RoboDK station: main2.rdk

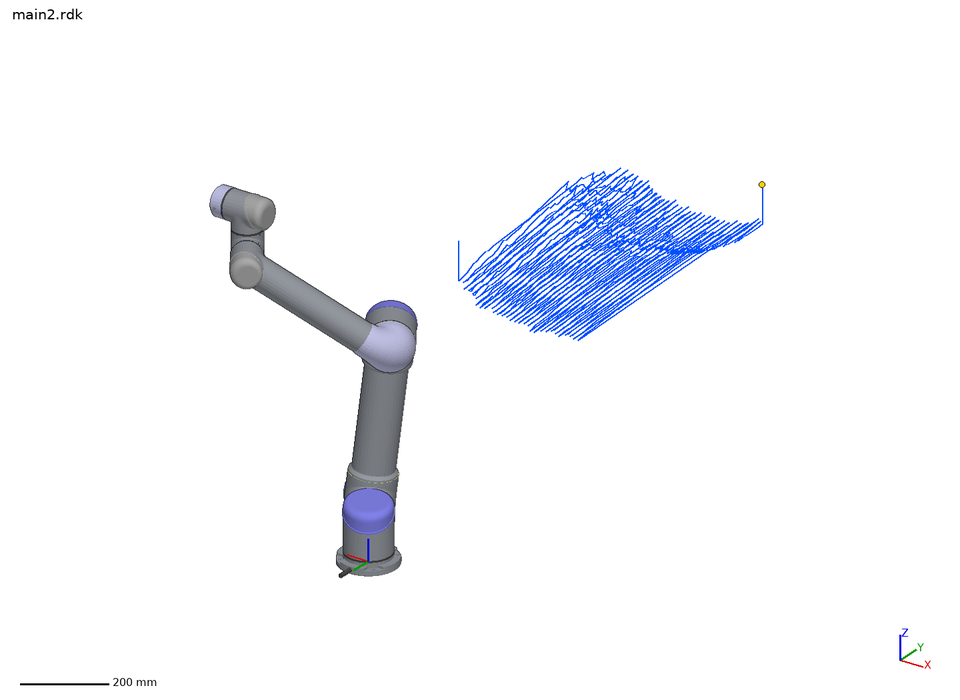
[picture v0: the station drawn from its stored meshes, robots at their saved joint values, targets as dots, program paths as lines]
Station main. Poses are relative to the parent item; angles as X-Y-Z fixed-axis rotations.
  - frame UR5 Base at (0, 0, 0) mm, rotated rx 0 ry 0 rz 180 deg
    - robot UR5: 6 axes, payload 5 kg, reach 850 mm, repeatability 0.1 mm, weight 18.4 kg
        modified DH rows (alpha deg, a mm, theta deg, d mm): 0, 0, 0, 89.2; 90, 0, 180, 0; 0, 425, 0, 0; 0, 392.43, 0, 109; -90, 0, 0, 93.65; 90, 0, 180, 82
        joint limits [-360, -360, -360, -360, -360, -360] to [360, 360, 360, 360, 360, 360]; home [0, -90, -90, 0, 90, 0]; saved at [33.979, -83.621, -61.636, -34.743, 56.021, -90]
  - frame Object at (-1200, -500, 400) mm, rotated rx -90 ry 0 rz -90 deg
    - object Curve at (0, 0, 0) mm
  - machining project AutoCurveFollow settings: rotZ(0) | rotX(0)*rotY(0) | rotz(0) | onStart | onPathStart | onApproach | onPoint | onRetract | onFinish | Extruder(%1) | default | default | OutOnMov(%1) | OutOffMov(%1) | onPathFinish | M_RunCode(%1)
  - program AutoCurveFollow (1423 instructions, listed below)
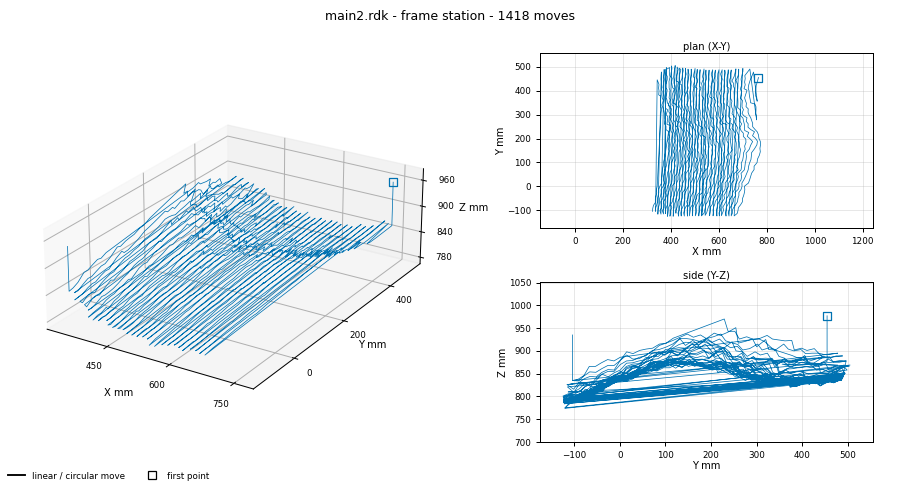
[picture p0: tool path of main2.rdk in frame station, 1418 of 1418 moves have a stored position in this frame; points joined in program order, loops and branches not executed]

--- program AutoCurveFollow (robot UR5) ---
  Set Ref.: UR5 Base
  Set Tool at (0, 0, 0) mm
  Set speed (1000.0 mm/s)
  MoveJ 1 to (-764.48, -454.56, 977) mm, rotated rx 180 ry 0 rz -90 deg; joints [-40.611, -86.577, -54.328, -39.095, 130.611, -90]
  MoveL 2 to (-764.48, -454.56, 977) mm, rotated rx 180 ry 0 rz -90 deg; joints [-40.611, -86.577, -54.328, -39.095, 130.611, -90]
  MoveL 3 to (-764.48, -454.56, 877) mm, rotated rx 180 ry 0 rz -90 deg; joints [-29.923, -94.985, -45.76, -39.255, 119.923, -90]
  MoveL 4 to (-764.48, -454.56, 877) mm, rotated rx 180 ry 0 rz -90 deg; joints [-29.923, -94.985, -45.76, -39.255, 119.923, -90]
  Set speed (50.0 mm/s)
  MoveL 5 to (-760.12, -438.29, 872) mm, rotated rx 180 ry 0 rz -90 deg; joints [-28.873, -93.22, -50.699, -36.081, 118.873, -90]
  MoveL 6 to (-754.89, -421.7, 866) mm, rotated rx 180 ry 0 rz -90 deg; joints [-27.622, -91.69, -55.258, -33.052, 117.622, -90]
  MoveL 7 to (-754.02, -407.65, 865) mm, rotated rx 180 ry 0 rz -90 deg; joints [-27.415, -90.512, -58.88, -30.609, 117.415, -90]
  MoveL 8 to (-752.27, -393.17, 863) mm, rotated rx 180 ry 0 rz -90 deg; joints [-27.002, -89.439, -62.378, -28.183, 117.002, -90]
  MoveL 9 to (-752.27, -379.64, 863) mm, rotated rx 180 ry 0 rz -90 deg; joints [-27.002, -88.514, -65.502, -25.984, 117.002, -90]
  MoveL 10 to (-756.63, -368.22, 868) mm, rotated rx 180 ry 0 rz -90 deg; joints [-28.038, -87.745, -68.081, -24.174, 118.038, -90]
  MoveL 11 to (-759.25, -355.84, 871) mm, rotated rx 180 ry 0 rz -90 deg; joints [-28.664, -87.014, -70.74, -22.246, 118.664, -90]
  MoveL 12 to (-743.88, -477.67, 869) mm, rotated rx 180 ry 0 rz -90 deg; joints [-26.18, -96.591, -39.404, -44.005, 116.18, -90]
  MoveL 13 to (-729.32, -441.6, 852) mm, rotated rx 180 ry 0 rz -90 deg; joints [-22.685, -92.557, -50.807, -36.636, 112.685, -90]
  MoveL 14 to (-724.19, -425.22, 846) mm, rotated rx 180 ry 0 rz -90 deg; joints [-21.483, -91.151, -55.197, -33.652, 111.483, -90]
  MoveL 15 to (-721.62, -410.5, 843) mm, rotated rx 180 ry 0 rz -90 deg; joints [-20.889, -89.985, -58.924, -31.091, 110.889, -90]
  MoveL 16 to (-725.04, -399.16, 847) mm, rotated rx 180 ry 0 rz -90 deg; joints [-21.682, -88.972, -61.84, -29.189, 111.682, -90]
  MoveL 17 to (-725.9, -386.34, 848) mm, rotated rx 180 ry 0 rz -90 deg; joints [-21.882, -88.028, -64.877, -27.095, 111.882, -90]
  MoveL 18 to (-727.61, -373.92, 850) mm, rotated rx 180 ry 0 rz -90 deg; joints [-22.282, -87.165, -67.716, -25.119, 112.282, -90]
  MoveL 19 to (-730.18, -361.86, 853) mm, rotated rx 180 ry 0 rz -90 deg; joints [-22.887, -86.368, -70.389, -23.243, 112.887, -90]
  MoveL 20 to (-731.89, -349.3, 855) mm, rotated rx 180 ry 0 rz -90 deg; joints [-23.292, -85.64, -73.039, -21.321, 113.292, -90]
  MoveL 21 to (-749.87, -344.14, 876) mm, rotated rx 180 ry 0 rz -90 deg; joints [-27.655, -84.997, -74.428, -20.575, 117.655, -90]
  MoveL 22 to (-754.15, -332.29, 881) mm, rotated rx 180 ry 0 rz -90 deg; joints [-28.72, -84.394, -76.805, -18.802, 118.72, -90]
  MoveL 23 to (-754.15, -318.48, 881) mm, rotated rx 180 ry 0 rz -90 deg; joints [-28.72, -83.813, -79.436, -16.751, 118.72, -90]
  MoveL 24 to (-753.29, -304.32, 880) mm, rotated rx 180 ry 0 rz -90 deg; joints [-28.506, -83.297, -82.034, -14.669, 118.506, -90]
  MoveL 25 to (-755.86, -291.51, 883) mm, rotated rx 180 ry 0 rz -90 deg; joints [-29.148, -82.862, -84.336, -12.802, 119.148, -90]
  MoveL 26 to (-756.72, -277.98, 884) mm, rotated rx 180 ry 0 rz -90 deg; joints [-29.363, -82.481, -86.682, -10.837, 119.363, -90]
  MoveL 27 to (-728.57, -490.16, 867) mm, rotated rx 180 ry 0 rz -90 deg; joints [-23.594, -97.07, -36.241, -46.688, 113.594, -90]
  MoveL 28 to (-707.56, -462.82, 842) mm, rotated rx 180 ry 0 rz -90 deg; joints [-18.545, -94.089, -45.181, -40.73, 108.545, -90]
  MoveL 29 to (-709.24, -450.69, 844) mm, rotated rx 180 ry 0 rz -90 deg; joints [-18.936, -92.582, -49.108, -38.31, 108.936, -90]
  MoveL 30 to (-706.72, -435.9, 841) mm, rotated rx 180 ry 0 rz -90 deg; joints [-18.351, -91.172, -53.282, -35.546, 108.351, -90]
  MoveL 31 to (-709.24, -424.22, 844) mm, rotated rx 180 ry 0 rz -90 deg; joints [-18.936, -89.957, -56.582, -33.46, 108.936, -90]
  MoveL 32 to (-704.2, -408.06, 838) mm, rotated rx 180 ry 0 rz -90 deg; joints [-17.77, -88.854, -60.455, -30.691, 107.77, -90]
  MoveL 33 to (-716.8, -401.99, 853) mm, rotated rx 180 ry 0 rz -90 deg; joints [-20.724, -87.803, -62.493, -29.704, 110.724, -90]
  MoveL 34 to (-711.76, -385.88, 847) mm, rotated rx 180 ry 0 rz -90 deg; joints [-19.527, -86.87, -66.047, -27.083, 109.527, -90]
  MoveL 35 to (-706.72, -369.96, 841) mm, rotated rx 180 ry 0 rz -90 deg; joints [-18.351, -86.096, -69.346, -24.557, 108.351, -90]
  MoveL 36 to (-710.08, -358.47, 845) mm, rotated rx 180 ry 0 rz -90 deg; joints [-19.133, -85.277, -71.925, -22.798, 109.133, -90]
  MoveL 37 to (-714.28, -347.26, 850) mm, rotated rx 180 ry 0 rz -90 deg; joints [-20.123, -84.502, -74.384, -21.115, 110.123, -90]
  MoveL 38 to (-712.6, -333.14, 848) mm, rotated rx 180 ry 0 rz -90 deg; joints [-19.725, -83.901, -77.109, -18.991, 109.725, -90]
  MoveL 39 to (-721.85, -324, 859) mm, rotated rx 180 ry 0 rz -90 deg; joints [-21.941, -83.141, -79.178, -17.681, 111.942, -90]
  MoveL 40 to (-721.01, -310.16, 858) mm, rotated rx 180 ry 0 rz -90 deg; joints [-21.737, -82.629, -81.727, -15.645, 111.737, -90]
  MoveL 41 to (-725.21, -298.44, 863) mm, rotated rx 180 ry 0 rz -90 deg; joints [-22.763, -82.079, -83.965, -13.956, 112.764, -90]
  MoveL 42 to (-731.93, -287.55, 871) mm, rotated rx 180 ry 0 rz -90 deg; joints [-24.432, -81.55, -86.044, -12.406, 114.432, -90]
  MoveL 43 to (-736.13, -275.46, 876) mm, rotated rx 180 ry 0 rz -90 deg; joints [-25.49, -81.125, -88.199, -10.676, 115.49, -90]
  MoveL 44 to (-740.33, -263.22, 881) mm, rotated rx 180 ry 0 rz -90 deg; joints [-26.56, -80.762, -90.313, -8.925, 116.56, -90]
  MoveL 45 to (-740.33, -249.4, 881) mm, rotated rx 180 ry 0 rz -90 deg; joints [-26.56, -80.505, -92.561, -6.934, 116.56, -90]
  MoveL 46 to (-749.58, -238.53, 892) mm, rotated rx 180 ry 0 rz -90 deg; joints [-28.949, -80.229, -94.384, -5.388, 118.949, -90]
  MoveL 47 to (-759.66, -227.56, 904) mm, rotated rx 180 ry 0 rz -90 deg; joints [-31.605, -80.079, -96.112, -3.809, 121.605, -90]
  MoveL 48 to (-764.7, -214.8, 910) mm, rotated rx 180 ry 0 rz -90 deg; joints [-32.949, -80.016, -98.029, -1.955, 122.949, -90]
  MoveL 49 to (-766.38, -200.97, 912) mm, rotated rx 180 ry 0 rz -90 deg; joints [-33.399, -79.998, -100.063, 0.061, 123.399, -90]
  MoveL 50 to (-772.27, -188.1, 919) mm, rotated rx 180 ry 0 rz -90 deg; joints [-34.98, -80.101, -101.858, 1.959, 124.98, -90]
  MoveL 51 to (-773.11, -173.88, 920) mm, rotated rx 180 ry 0 rz -90 deg; joints [-35.206, -80.218, -103.843, 4.06, 125.206, -90]
  MoveL 52 to (-770.59, -158.93, 917) mm, rotated rx 180 ry 0 rz -90 deg; joints [-34.527, -80.368, -105.912, 6.279, 124.527, -90]
  MoveL 53 to (-772.27, -144.87, 919) mm, rotated rx 180 ry 0 rz -90 deg; joints [-34.98, -80.645, -107.755, 8.4, 124.98, -90]
  MoveL 54 to (-768.07, -129.75, 914) mm, rotated rx 180 ry 0 rz -90 deg; joints [-33.849, -80.946, -109.745, 10.691, 123.849, -90]
  MoveL 55 to (-760.5, -114.28, 905) mm, rotated rx 180 ry 0 rz -90 deg; joints [-31.828, -81.351, -111.718, 13.069, 121.829, -90]
  MoveL 56 to (-758.82, -99.87, 903) mm, rotated rx 180 ry 0 rz -90 deg; joints [-31.382, -81.864, -113.459, 15.323, 121.382, -90]
  MoveL 57 to (-746.22, -84.28, 888) mm, rotated rx 180 ry 0 rz -90 deg; joints [-28.075, -82.59, -115.218, 17.808, 118.075, -90]
  MoveL 58 to (-746.22, -70.36, 888) mm, rotated rx 180 ry 0 rz -90 deg; joints [-28.075, -83.267, -116.786, 20.053, 118.075, -90]
  MoveL 59 to (-736.13, -55.67, 876) mm, rotated rx 180 ry 0 rz -90 deg; joints [-25.49, -84.254, -118.225, 22.479, 115.491, -90]
  MoveL 60 to (-731.93, -41.69, 871) mm, rotated rx 180 ry 0 rz -90 deg; joints [-24.432, -85.223, -119.589, 24.812, 114.432, -90]
  MoveL 61 to (-727.73, -27.87, 866) mm, rotated rx 180 ry 0 rz -90 deg; joints [-23.386, -86.291, -120.861, 27.152, 113.386, -90]
  MoveL 62 to (-722.69, -14.2, 860) mm, rotated rx 180 ry 0 rz -90 deg; joints [-22.146, -87.486, -122.014, 29.5, 112.146, -90]
  MoveL 63 to (-705.88, -0.69, 840) mm, rotated rx 180 ry 0 rz -90 deg; joints [-18.157, -89.326, -122.532, 31.857, 108.157, -90]
  MoveL 64 to (-707.56, 12.51, 842) mm, rotated rx 180 ry 0 rz -90 deg; joints [-18.546, -90.399, -123.761, 34.159, 108.546, -90]
  MoveL 65 to (-705.88, 25.65, 840) mm, rotated rx 180 ry 0 rz -90 deg; joints [-18.157, -91.722, -124.757, 36.479, 108.157, -90]
  MoveL 66 to (-702.52, 38.64, 836) mm, rotated rx 180 ry 0 rz -90 deg; joints [-17.387, -93.202, -125.584, 38.786, 107.387, -90]
  MoveL 67 to (-697.48, 51.38, 830) mm, rotated rx 180 ry 0 rz -90 deg; joints [-16.25, -94.833, -126.217, 41.05, 106.25, -90]
  MoveL 68 to (-697.48, 64.39, 830) mm, rotated rx 180 ry 0 rz -90 deg; joints [-16.25, -96.303, -127.104, 43.408, 106.25, -90]
  MoveL 69 to (-689.91, 76.57, 821) mm, rotated rx 180 ry 0 rz -90 deg; joints [-14.586, -98.171, -127.371, 45.542, 104.586, -90]
  MoveL 70 to (-680.67, 88.24, 810) mm, rotated rx 180 ry 0 rz -90 deg; joints [-12.622, -100.166, -127.353, 47.52, 102.622, -90]
  MoveL 71 to (-678.99, 100.7, 808) mm, rotated rx 180 ry 0 rz -90 deg; joints [-12.274, -101.861, -127.879, 49.74, 102.274, -90]
  MoveL 72 to (-675.63, 112.81, 804) mm, rotated rx 180 ry 0 rz -90 deg; joints [-11.584, -103.674, -128.178, 51.851, 101.584, -90]
  MoveL 73 to (-663.02, 123.08, 789) mm, rotated rx 180 ry 0 rz -90 deg; joints [-9.09, -105.869, -127.452, 53.321, 99.09, -90]
  MoveL 74 to (-699.31, -492.72, 848) mm, rotated rx 180 ry 0 rz -90 deg; joints [-17.48, -96.856, -35.95, -47.194, 107.48, -90]
  MoveL 75 to (-699.31, -479.42, 848) mm, rotated rx 180 ry 0 rz -90 deg; joints [-17.48, -94.798, -41.109, -44.093, 107.48, -90]
  MoveL 76 to (-695.18, -463.37, 843) mm, rotated rx 180 ry 0 rz -90 deg; joints [-16.507, -92.936, -46.33, -40.735, 106.507, -90]
  MoveL 77 to (-691.88, -448.02, 839) mm, rotated rx 180 ry 0 rz -90 deg; joints [-15.741, -91.394, -50.848, -37.758, 105.741, -90]
  MoveL 78 to (-693.53, -435.9, 841) mm, rotated rx 180 ry 0 rz -90 deg; joints [-16.123, -90.065, -54.405, -35.53, 106.123, -90]
  MoveL 79 to (-694.36, -423.21, 842) mm, rotated rx 180 ry 0 rz -90 deg; joints [-16.315, -88.852, -57.848, -33.3, 106.315, -90]
  MoveL 80 to (-688.58, -406.6, 835) mm, rotated rx 180 ry 0 rz -90 deg; joints [-14.985, -87.834, -61.685, -30.48, 104.985, -90]
  MoveL 81 to (-693.53, -396.33, 841) mm, rotated rx 180 ry 0 rz -90 deg; joints [-16.123, -86.765, -64.417, -28.818, 106.123, -90]
  MoveL 82 to (-691.88, -382.24, 839) mm, rotated rx 180 ry 0 rz -90 deg; joints [-15.741, -85.896, -67.543, -26.561, 105.741, -90]
  MoveL 83 to (-689.41, -367.76, 836) mm, rotated rx 180 ry 0 rz -90 deg; joints [-15.173, -85.149, -70.561, -24.291, 105.173, -90]
  MoveL 84 to (-697.66, -358.89, 846) mm, rotated rx 180 ry 0 rz -90 deg; joints [-17.089, -84.166, -72.848, -22.986, 107.089, -90]
  MoveL 85 to (-696.01, -344.81, 844) mm, rotated rx 180 ry 0 rz -90 deg; joints [-16.701, -83.52, -75.63, -20.85, 106.701, -90]
  MoveL 86 to (-696.01, -331.57, 844) mm, rotated rx 180 ry 0 rz -90 deg; joints [-16.701, -82.898, -78.222, -18.88, 106.701, -90]
  MoveL 87 to (-701.78, -320.98, 851) mm, rotated rx 180 ry 0 rz -90 deg; joints [-18.072, -82.14, -80.495, -17.365, 108.072, -90]
  MoveL 88 to (-696.01, -305.1, 844) mm, rotated rx 180 ry 0 rz -90 deg; joints [-16.701, -81.844, -83.158, -14.998, 106.701, -90]
  MoveL 89 to (-703.43, -294.98, 853) mm, rotated rx 180 ry 0 rz -90 deg; joints [-18.469, -81.115, -85.292, -13.593, 108.469, -90]
  MoveL 90 to (-716.62, -286.89, 869) mm, rotated rx 180 ry 0 rz -90 deg; joints [-21.738, -80.305, -87.169, -12.525, 111.738, -90]
  MoveL 91 to (-713.32, -272, 865) mm, rotated rx 180 ry 0 rz -90 deg; joints [-20.906, -80.032, -89.608, -10.36, 110.906, -90]
  MoveL 92 to (-721.57, -261.42, 875) mm, rotated rx 180 ry 0 rz -90 deg; joints [-23.002, -79.5, -91.603, -8.897, 113.002, -90]
  MoveL 93 to (-720.75, -247.42, 874) mm, rotated rx 180 ry 0 rz -90 deg; joints [-22.79, -79.267, -93.853, -6.88, 112.79, -90]
  MoveL 94 to (-732.29, -237.46, 888) mm, rotated rx 180 ry 0 rz -90 deg; joints [-25.806, -78.816, -95.674, -5.51, 115.806, -90]
  MoveL 95 to (-747.96, -228.32, 907) mm, rotated rx 180 ry 0 rz -90 deg; joints [-30.045, -78.523, -97.244, -4.233, 120.045, -90]
  MoveL 96 to (-739.71, -211.73, 897) mm, rotated rx 180 ry 0 rz -90 deg; joints [-27.795, -78.47, -99.71, -1.82, 117.795, -90]
  MoveL 97 to (-752.08, -200.97, 912) mm, rotated rx 180 ry 0 rz -90 deg; joints [-31.183, -78.371, -101.359, -0.27, 121.183, -90]
  MoveL 98 to (-760.33, -188.72, 922) mm, rotated rx 180 ry 0 rz -90 deg; joints [-33.482, -78.436, -103.098, 1.534, 123.482, -90]
  MoveL 99 to (-757.86, -173.69, 919) mm, rotated rx 180 ry 0 rz -90 deg; joints [-32.79, -78.511, -105.236, 3.746, 122.79, -90]
  MoveL 100 to (-747.96, -157.2, 907) mm, rotated rx 180 ry 0 rz -90 deg; joints [-30.045, -78.692, -107.51, 6.202, 120.045, -90]
  MoveL 101 to (-735.59, -140.61, 892) mm, rotated rx 180 ry 0 rz -90 deg; joints [-26.686, -79.13, -109.607, 8.737, 116.686, -90]
  MoveL 102 to (-734.77, -126.48, 891) mm, rotated rx 180 ry 0 rz -90 deg; joints [-26.465, -79.492, -111.412, 10.905, 116.465, -90]
  MoveL 103 to (-733.12, -112.26, 889) mm, rotated rx 180 ry 0 rz -90 deg; joints [-26.026, -79.956, -113.164, 13.12, 116.026, -90]
  MoveL 104 to (-727.34, -97.54, 882) mm, rotated rx 180 ry 0 rz -90 deg; joints [-24.501, -80.63, -114.834, 15.464, 114.501, -90]
  MoveL 105 to (-723.22, -83.24, 877) mm, rotated rx 180 ry 0 rz -90 deg; joints [-23.428, -81.364, -116.409, 17.773, 113.428, -90]
  MoveL 106 to (-721.57, -69.33, 875) mm, rotated rx 180 ry 0 rz -90 deg; joints [-23.002, -82.101, -117.941, 20.042, 113.002, -90]
  MoveL 107 to (-715.8, -55.16, 868) mm, rotated rx 180 ry 0 rz -90 deg; joints [-21.529, -83.102, -119.308, 22.411, 111.529, -90]
  MoveL 108 to (-710.03, -41.22, 861) mm, rotated rx 180 ry 0 rz -90 deg; joints [-20.084, -84.219, -120.559, 24.779, 110.084, -90]
  MoveL 109 to (-703.43, -27.46, 853) mm, rotated rx 180 ry 0 rz -90 deg; joints [-18.469, -85.494, -121.657, 27.151, 108.469, -90]
  MoveL 110 to (-695.18, -13.92, 843) mm, rotated rx 180 ry 0 rz -90 deg; joints [-16.507, -86.983, -122.535, 29.517, 106.507, -90]
  MoveL 111 to (-696.01, -0.7, 844) mm, rotated rx 180 ry 0 rz -90 deg; joints [-16.701, -88.019, -123.799, 31.818, 106.701, -90]
  MoveL 112 to (-691.88, 12.46, 839) mm, rotated rx 180 ry 0 rz -90 deg; joints [-15.741, -89.438, -124.712, 34.15, 105.741, -90]
  MoveL 113 to (-682.81, 25.28, 828) mm, rotated rx 180 ry 0 rz -90 deg; joints [-13.688, -91.25, -125.178, 36.429, 103.688, -90]
  MoveL 114 to (-682.81, 38.27, 828) mm, rotated rx 180 ry 0 rz -90 deg; joints [-13.688, -92.565, -126.196, 38.761, 103.688, -90]
  MoveL 115 to (-678.69, 50.94, 823) mm, rotated rx 180 ry 0 rz -90 deg; joints [-12.781, -94.212, -126.824, 41.036, 102.781, -90]
  MoveL 116 to (-677.04, 63.69, 821) mm, rotated rx 180 ry 0 rz -90 deg; joints [-12.423, -95.776, -127.575, 43.35, 102.423, -90]
  MoveL 117 to (-669.62, 75.73, 812) mm, rotated rx 180 ry 0 rz -90 deg; joints [-10.847, -97.735, -127.725, 45.46, 100.848, -90]
  MoveL 118 to (-661.37, 87.37, 802) mm, rotated rx 180 ry 0 rz -90 deg; joints [-9.162, -99.784, -127.653, 47.437, 99.162, -90]
  MoveL 119 to (-655.6, 99.08, 795) mm, rotated rx 180 ry 0 rz -90 deg; joints [-8.022, -101.716, -127.709, 49.425, 98.022, -90]
  MoveL 120 to (-655.6, 111.54, 795) mm, rotated rx 180 ry 0 rz -90 deg; joints [-8.022, -103.363, -128.317, 51.68, 98.022, -90]
  MoveL 121 to (-650.65, 123.08, 789) mm, rotated rx 180 ry 0 rz -90 deg; joints [-7.072, -105.302, -128.296, 53.598, 97.072, -90]
  MoveL 122 to (-681.96, -489.81, 843) mm, rotated rx 180 ry 0 rz -90 deg; joints [-14.19, -95.436, -38.23, -46.334, 104.19, -90]
  MoveL 123 to (-681.96, -476.59, 843) mm, rotated rx 180 ry 0 rz -90 deg; joints [-14.19, -93.507, -43.112, -43.381, 104.19, -90]
  MoveL 124 to (-679.54, -461.73, 840) mm, rotated rx 180 ry 0 rz -90 deg; joints [-13.624, -91.807, -47.841, -40.351, 103.624, -90]
  MoveL 125 to (-670.64, -442.68, 829) mm, rotated rx 180 ry 0 rz -90 deg; joints [-11.607, -90.407, -52.836, -36.758, 101.608, -90]
  MoveL 126 to (-674.68, -432.27, 834) mm, rotated rx 180 ry 0 rz -90 deg; joints [-12.513, -89.085, -56.024, -34.891, 102.513, -90]
  MoveL 127 to (-677.92, -421.2, 838) mm, rotated rx 180 ry 0 rz -90 deg; joints [-13.251, -87.863, -59.151, -32.986, 103.251, -90]
  MoveL 128 to (-677.92, -408.06, 838) mm, rotated rx 180 ry 0 rz -90 deg; joints [-13.251, -86.791, -62.419, -30.79, 103.251, -90]
  MoveL 129 to (-675.49, -393.51, 835) mm, rotated rx 180 ry 0 rz -90 deg; joints [-12.697, -85.886, -65.697, -28.417, 102.697, -90]
  MoveL 130 to (-676.3, -380.87, 836) mm, rotated rx 180 ry 0 rz -90 deg; joints [-12.881, -84.976, -68.597, -26.427, 102.881, -90]
  MoveL 131 to (-677.92, -368.64, 838) mm, rotated rx 180 ry 0 rz -90 deg; joints [-13.251, -84.107, -71.345, -24.548, 103.251, -90]
  MoveL 132 to (-678.73, -355.92, 839) mm, rotated rx 180 ry 0 rz -90 deg; joints [-13.437, -83.333, -74.045, -22.622, 103.437, -90]
  MoveL 133 to (-678.73, -342.77, 839) mm, rotated rx 180 ry 0 rz -90 deg; joints [-13.437, -82.657, -76.692, -20.651, 103.437, -90]
  MoveL 134 to (-677.92, -329.22, 838) mm, rotated rx 180 ry 0 rz -90 deg; joints [-13.251, -82.085, -79.277, -18.638, 103.251, -90]
  MoveL 135 to (-687.63, -320.6, 850) mm, rotated rx 180 ry 0 rz -90 deg; joints [-15.534, -81.087, -81.431, -17.481, 105.534, -90]
  MoveL 136 to (-690.05, -308.36, 853) mm, rotated rx 180 ry 0 rz -90 deg; joints [-16.121, -80.467, -83.805, -15.728, 106.121, -90]
  MoveL 137 to (-690.05, -294.98, 853) mm, rotated rx 180 ry 0 rz -90 deg; joints [-16.121, -80.006, -86.198, -13.796, 106.121, -90]
  MoveL 138 to (-699.76, -285.57, 865) mm, rotated rx 180 ry 0 rz -90 deg; joints [-18.53, -79.193, -88.26, -12.547, 108.53, -90]
  MoveL 139 to (-702.19, -272.94, 868) mm, rotated rx 180 ry 0 rz -90 deg; joints [-19.148, -78.733, -90.504, -10.763, 109.148, -90]
  MoveL 140 to (-705.42, -260.53, 872) mm, rotated rx 180 ry 0 rz -90 deg; joints [-19.981, -78.299, -92.683, -9.018, 109.981, -90]
  MoveL 141 to (-706.23, -247.14, 873) mm, rotated rx 180 ry 0 rz -90 deg; joints [-20.19, -78.01, -94.882, -7.108, 110.19, -90]
  MoveL 142 to (-707.04, -233.71, 874) mm, rotated rx 180 ry 0 rz -90 deg; joints [-20.401, -77.781, -97.03, -5.189, 110.401, -90]
  MoveL 143 to (-724.03, -225.3, 895) mm, rotated rx 180 ry 0 rz -90 deg; joints [-24.961, -77.124, -98.765, -4.111, 114.961, -90]
  MoveL 144 to (-717.56, -209.37, 887) mm, rotated rx 180 ry 0 rz -90 deg; joints [-23.193, -77.19, -101.043, -1.767, 113.193, -90]
  MoveL 145 to (-729.69, -198.77, 902) mm, rotated rx 180 ry 0 rz -90 deg; joints [-26.535, -76.867, -102.836, -0.297, 116.535, -90]
  MoveL 146 to (-740.21, -187.28, 915) mm, rotated rx 180 ry 0 rz -90 deg; joints [-29.52, -76.763, -104.591, 1.354, 119.521, -90]
  MoveL 147 to (-731.31, -170.86, 904) mm, rotated rx 180 ry 0 rz -90 deg; joints [-26.989, -76.959, -106.844, 3.803, 116.989, -90]
  MoveL 148 to (-726.46, -155.64, 898) mm, rotated rx 180 ry 0 rz -90 deg; joints [-25.632, -77.237, -108.864, 6.101, 115.632, -90]
  MoveL 149 to (-712.7, -138.88, 881) mm, rotated rx 180 ry 0 rz -90 deg; joints [-21.892, -77.959, -110.779, 8.738, 111.892, -90]
  MoveL 150 to (-714.32, -125.35, 883) mm, rotated rx 180 ry 0 rz -90 deg; joints [-22.323, -78.232, -112.573, 10.805, 112.323, -90]
  MoveL 151 to (-712.7, -111.25, 881) mm, rotated rx 180 ry 0 rz -90 deg; joints [-21.892, -78.72, -114.296, 13.017, 111.892, -90]
  MoveL 152 to (-709.47, -96.99, 877) mm, rotated rx 180 ry 0 rz -90 deg; joints [-21.036, -79.371, -115.931, 15.302, 111.036, -90]
  MoveL 153 to (-707.85, -83.05, 875) mm, rotated rx 180 ry 0 rz -90 deg; joints [-20.612, -80.037, -117.522, 17.559, 110.612, -90]
  MoveL 154 to (-705.42, -69.09, 872) mm, rotated rx 180 ry 0 rz -90 deg; joints [-19.981, -80.834, -119.028, 19.862, 109.981, -90]
  MoveL 155 to (-691.67, -54.34, 855) mm, rotated rx 180 ry 0 rz -90 deg; joints [-16.515, -82.418, -120.022, 22.44, 106.515, -90]
  MoveL 156 to (-694.1, -41.07, 858) mm, rotated rx 180 ry 0 rz -90 deg; joints [-17.113, -83.101, -121.554, 24.654, 107.113, -90]
  MoveL 157 to (-691.67, -27.52, 855) mm, rotated rx 180 ry 0 rz -90 deg; joints [-16.515, -84.189, -122.808, 26.997, 106.515, -90]
  MoveL 158 to (-682.77, -13.93, 844) mm, rotated rx 180 ry 0 rz -90 deg; joints [-14.38, -85.816, -123.607, 29.423, 104.38, -90]
  MoveL 159 to (-683.58, -0.7, 845) mm, rotated rx 180 ry 0 rz -90 deg; joints [-14.57, -86.858, -124.894, 31.752, 104.57, -90]
  MoveL 160 to (-679.54, 12.48, 840) mm, rotated rx 180 ry 0 rz -90 deg; joints [-13.624, -88.329, -125.795, 34.124, 103.624, -90]
  MoveL 161 to (-666.59, 25.16, 824) mm, rotated rx 180 ry 0 rz -90 deg; joints [-10.72, -90.55, -125.871, 36.421, 100.72, -90]
  MoveL 162 to (-669.02, 38.22, 827) mm, rotated rx 180 ry 0 rz -90 deg; joints [-11.25, -91.691, -127.107, 38.798, 101.25, -90]
  MoveL 163 to (-660.93, 50.57, 817) mm, rotated rx 180 ry 0 rz -90 deg; joints [-9.508, -93.69, -127.326, 41.016, 99.508, -90]
  MoveL 164 to (-659.31, 63.23, 815) mm, rotated rx 180 ry 0 rz -90 deg; joints [-9.168, -95.272, -128.057, 43.329, 99.168, -90]
  MoveL 165 to (-653.65, 75.36, 808) mm, rotated rx 180 ry 0 rz -90 deg; joints [-8.002, -97.2, -128.29, 45.49, 98.002, -90]
  MoveL 166 to (-647.18, 87.16, 800) mm, rotated rx 180 ry 0 rz -90 deg; joints [-6.712, -99.221, -128.319, 47.54, 96.712, -90]
  MoveL 167 to (-641.51, 98.83, 793) mm, rotated rx 180 ry 0 rz -90 deg; joints [-5.621, -101.21, -128.326, 49.536, 95.621, -90]
  MoveL 168 to (-638.28, 110.7, 789) mm, rotated rx 180 ry 0 rz -90 deg; joints [-5.013, -103.065, -128.536, 51.601, 95.013, -90]
  MoveL 169 to (-641.51, 123.7, 793) mm, rotated rx 180 ry 0 rz -90 deg; joints [-5.621, -104.598, -129.489, 54.086, 95.621, -90]
  MoveL 170 to (-670.33, -490.98, 845) mm, rotated rx 180 ry 0 rz -90 deg; joints [-12.161, -94.36, -39.205, -46.436, 102.161, -90]
  MoveL 171 to (-667.16, -475.46, 841) mm, rotated rx 180 ry 0 rz -90 deg; joints [-11.42, -92.42, -44.509, -43.071, 101.42, -90]
  MoveL 172 to (-663.19, -459.53, 836) mm, rotated rx 180 ry 0 rz -90 deg; joints [-10.513, -90.806, -49.295, -39.899, 100.513, -90]
  MoveL 173 to (-653.67, -440.01, 824) mm, rotated rx 180 ry 0 rz -90 deg; joints [-8.414, -89.587, -54.14, -36.273, 98.414, -90]
  MoveL 174 to (-660.02, -431.23, 832) mm, rotated rx 180 ry 0 rz -90 deg; joints [-9.8, -88.189, -57.077, -34.735, 99.8, -90]
  MoveL 175 to (-660.02, -418.19, 832) mm, rotated rx 180 ry 0 rz -90 deg; joints [-9.8, -87.05, -60.442, -32.509, 99.8, -90]
  MoveL 176 to (-664.78, -408.06, 838) mm, rotated rx 180 ry 0 rz -90 deg; joints [-10.873, -85.845, -63.289, -30.866, 100.873, -90]
  MoveL 177 to (-662.4, -393.51, 835) mm, rotated rx 180 ry 0 rz -90 deg; joints [-10.333, -84.964, -66.528, -28.508, 100.333, -90]
  MoveL 178 to (-663.19, -380.87, 836) mm, rotated rx 180 ry 0 rz -90 deg; joints [-10.513, -84.05, -69.416, -26.534, 100.513, -90]
  MoveL 179 to (-663.19, -367.76, 836) mm, rotated rx 180 ry 0 rz -90 deg; joints [-10.513, -83.244, -72.236, -24.52, 100.513, -90]
  MoveL 180 to (-663.98, -355.07, 837) mm, rotated rx 180 ry 0 rz -90 deg; joints [-10.693, -82.467, -74.919, -22.613, 100.693, -90]
  MoveL 181 to (-663.98, -341.95, 837) mm, rotated rx 180 ry 0 rz -90 deg; joints [-10.693, -81.796, -77.546, -20.659, 100.693, -90]
  MoveL 182 to (-668.74, -331.18, 843) mm, rotated rx 180 ry 0 rz -90 deg; joints [-11.789, -80.921, -79.941, -19.138, 101.789, -90]
  MoveL 183 to (-671.12, -319.09, 846) mm, rotated rx 180 ry 0 rz -90 deg; joints [-12.348, -80.226, -82.365, -17.409, 102.348, -90]
  MoveL 184 to (-681.44, -297.06, 859) mm, rotated rx 180 ry 0 rz -90 deg; joints [-14.849, -78.698, -86.924, -14.378, 104.85, -90]
  MoveL 185 to (-686.99, -285.9, 866) mm, rotated rx 180 ry 0 rz -90 deg; joints [-16.25, -78.004, -89.138, -12.858, 106.25, -90]
  MoveL 186 to (-686.99, -272.32, 866) mm, rotated rx 180 ry 0 rz -90 deg; joints [-16.25, -77.627, -91.453, -10.92, 106.25, -90]
  MoveL 187 to (-694.13, -261.42, 875) mm, rotated rx 180 ry 0 rz -90 deg; joints [-18.106, -76.974, -93.564, -9.462, 108.106, -90]
  MoveL 188 to (-686.99, -245.16, 866) mm, rotated rx 180 ry 0 rz -90 deg; joints [-16.25, -77.054, -95.904, -7.042, 106.25, -90]
  MoveL 189 to (-691.75, -233.18, 872) mm, rotated rx 180 ry 0 rz -90 deg; joints [-17.481, -76.605, -98, -5.394, 107.481, -90]
  MoveL 190 to (-701.27, -222.53, 884) mm, rotated rx 180 ry 0 rz -90 deg; joints [-20.02, -76.014, -100, -3.986, 110.02, -90]
  MoveL 191 to (-701.27, -208.66, 884) mm, rotated rx 180 ry 0 rz -90 deg; joints [-20.02, -75.915, -102.1, -1.985, 110.02, -90]
  MoveL 192 to (-711.58, -197.67, 897) mm, rotated rx 180 ry 0 rz -90 deg; joints [-22.882, -75.483, -104.023, -0.495, 112.882, -90]
  MoveL 193 to (-712.37, -183.81, 898) mm, rotated rx 180 ry 0 rz -90 deg; joints [-23.107, -75.475, -106.053, 1.527, 113.107, -90]
  MoveL 194 to (-706.82, -168.4, 891) mm, rotated rx 180 ry 0 rz -90 deg; joints [-21.547, -75.774, -108.086, 3.859, 111.547, -90]
  MoveL 195 to (-709.2, -154.95, 894) mm, rotated rx 180 ry 0 rz -90 deg; joints [-22.211, -75.846, -110.004, 5.85, 112.211, -90]
  MoveL 196 to (-702.06, -139.51, 885) mm, rotated rx 180 ry 0 rz -90 deg; joints [-20.236, -76.413, -111.857, 8.27, 110.236, -90]
  MoveL 197 to (-701.27, -125.49, 884) mm, rotated rx 180 ry 0 rz -90 deg; joints [-20.02, -76.783, -113.655, 10.438, 110.02, -90]
  MoveL 198 to (-698.89, -111.25, 881) mm, rotated rx 180 ry 0 rz -90 deg; joints [-19.375, -77.322, -115.373, 12.694, 109.375, -90]
  MoveL 199 to (-692.54, -96.55, 873) mm, rotated rx 180 ry 0 rz -90 deg; joints [-17.688, -78.196, -116.916, 15.112, 107.688, -90]
  MoveL 200 to (-694.13, -83.05, 875) mm, rotated rx 180 ry 0 rz -90 deg; joints [-18.106, -78.679, -118.595, 17.274, 108.106, -90]
  MoveL 201 to (-691.75, -69.09, 872) mm, rotated rx 180 ry 0 rz -90 deg; joints [-17.481, -79.5, -120.1, 19.6, 107.481, -90]
  MoveL 202 to (-677.47, -54.27, 854) mm, rotated rx 180 ry 0 rz -90 deg; joints [-13.872, -81.295, -120.969, 22.264, 103.872, -90]
  MoveL 203 to (-680.64, -41.07, 858) mm, rotated rx 180 ry 0 rz -90 deg; joints [-14.652, -81.89, -122.576, 24.466, 104.653, -90]
  MoveL 204 to (-677.47, -27.49, 854) mm, rotated rx 180 ry 0 rz -90 deg; joints [-13.872, -83.072, -123.781, 26.852, 103.872, -90]
  MoveL 205 to (-671.12, -13.96, 846) mm, rotated rx 180 ry 0 rz -90 deg; joints [-12.348, -84.606, -124.686, 29.292, 102.348, -90]
  MoveL 206 to (-667.16, -0.69, 841) mm, rotated rx 180 ry 0 rz -90 deg; joints [-11.42, -86.045, -125.643, 31.688, 101.42, -90]
  MoveL 207 to (-664.78, 12.45, 838) mm, rotated rx 180 ry 0 rz -90 deg; joints [-10.873, -87.439, -126.637, 34.076, 100.873, -90]
  MoveL 208 to (-656.84, 25.28, 828) mm, rotated rx 180 ry 0 rz -90 deg; joints [-9.101, -89.389, -127.054, 36.442, 99.101, -90]
  MoveL 209 to (-655.26, 38.18, 826) mm, rotated rx 180 ry 0 rz -90 deg; joints [-8.756, -90.871, -127.944, 38.815, 98.756, -90]
  MoveL 210 to (-647.32, 50.51, 816) mm, rotated rx 180 ry 0 rz -90 deg; joints [-7.076, -92.963, -128.102, 41.065, 97.076, -90]
  MoveL 211 to (-642.56, 62.84, 810) mm, rotated rx 180 ry 0 rz -90 deg; joints [-6.105, -94.839, -128.469, 43.308, 96.105, -90]
  MoveL 212 to (-637.01, 74.89, 803) mm, rotated rx 180 ry 0 rz -90 deg; joints [-5.007, -96.827, -128.637, 45.464, 95.007, -90]
  MoveL 213 to (-630.67, 86.61, 795) mm, rotated rx 180 ry 0 rz -90 deg; joints [-3.795, -98.909, -128.591, 47.5, 93.795, -90]
  MoveL 214 to (-629.08, 98.83, 793) mm, rotated rx 180 ry 0 rz -90 deg; joints [-3.5, -100.648, -129.067, 49.715, 93.5, -90]
  MoveL 215 to (-626.7, 110.84, 790) mm, rotated rx 180 ry 0 rz -90 deg; joints [-3.062, -102.491, -129.365, 51.856, 93.062, -90]
  MoveL 216 to (-629.08, 123.7, 793) mm, rotated rx 180 ry 0 rz -90 deg; joints [-3.5, -104.081, -130.242, 54.323, 93.5, -90]
  MoveL 217 to (-650.86, -486.33, 837) mm, rotated rx 180 ry 0 rz -90 deg; joints [-8.246, -93.226, -41.43, -45.344, 98.246, -90]
  MoveL 218 to (-647.75, -470.94, 833) mm, rotated rx 180 ry 0 rz -90 deg; joints [-7.554, -91.47, -46.404, -42.127, 97.554, -90]
  MoveL 219 to (-648.53, -458.43, 834) mm, rotated rx 180 ry 0 rz -90 deg; joints [-7.726, -89.916, -50.402, -39.683, 97.726, -90]
  MoveL 220 to (-643.08, -441.61, 827) mm, rotated rx 180 ry 0 rz -90 deg; joints [-6.542, -88.69, -54.729, -36.581, 96.542, -90]
  MoveL 221 to (-645.41, -430.2, 830) mm, rotated rx 180 ry 0 rz -90 deg; joints [-7.044, -87.384, -58.024, -34.592, 97.044, -90]
  MoveL 222 to (-652.41, -421.71, 839) mm, rotated rx 180 ry 0 rz -90 deg; joints [-8.596, -85.991, -60.806, -33.203, 98.596, -90]
  MoveL 223 to (-650.86, -407.58, 837) mm, rotated rx 180 ry 0 rz -90 deg; joints [-8.246, -84.991, -64.139, -30.87, 98.246, -90]
  MoveL 224 to (-646.97, -392.09, 832) mm, rotated rx 180 ry 0 rz -90 deg; joints [-7.383, -84.218, -67.422, -28.36, 97.383, -90]
  MoveL 225 to (-647.75, -379.5, 833) mm, rotated rx 180 ry 0 rz -90 deg; joints [-7.554, -83.308, -70.282, -26.41, 97.554, -90]
  MoveL 226 to (-648.53, -366.88, 834) mm, rotated rx 180 ry 0 rz -90 deg; joints [-7.726, -82.466, -73.04, -24.494, 97.726, -90]
  MoveL 227 to (-653.97, -356.77, 841) mm, rotated rx 180 ry 0 rz -90 deg; joints [-8.95, -81.407, -75.536, -23.057, 98.95, -90]
  MoveL 228 to (-650.86, -341.95, 837) mm, rotated rx 180 ry 0 rz -90 deg; joints [-8.246, -80.917, -78.272, -20.812, 98.246, -90]
  MoveL 229 to (-653.19, -330, 840) mm, rotated rx 180 ry 0 rz -90 deg; joints [-8.773, -80.149, -80.75, -19.101, 98.773, -90]
  MoveL 230 to (-657.86, -319.09, 846) mm, rotated rx 180 ry 0 rz -90 deg; joints [-9.85, -79.279, -83.121, -17.601, 99.85, -90]
  MoveL 231 to (-653.97, -304.02, 841) mm, rotated rx 180 ry 0 rz -90 deg; joints [-8.95, -79.035, -85.608, -15.357, 98.95, -90]
  MoveL 232 to (-661.74, -294.29, 851) mm, rotated rx 180 ry 0 rz -90 deg; joints [-10.771, -78.041, -87.85, -14.109, 100.771, -90]
  MoveL 233 to (-668.74, -283.92, 860) mm, rotated rx 180 ry 0 rz -90 deg; joints [-12.481, -77.171, -90.069, -12.76, 102.481, -90]
  MoveL 234 to (-663.3, -268.23, 853) mm, rotated rx 180 ry 0 rz -90 deg; joints [-11.145, -77.168, -92.409, -10.423, 101.145, -90]
  MoveL 235 to (-670.3, -257.54, 862) mm, rotated rx 180 ry 0 rz -90 deg; joints [-12.87, -76.383, -94.58, -9.037, 102.87, -90]
  MoveL 236 to (-677.3, -246.57, 871) mm, rotated rx 180 ry 0 rz -90 deg; joints [-14.663, -75.677, -96.719, -7.605, 104.663, -90]
  MoveL 237 to (-673.41, -231.58, 866) mm, rotated rx 180 ry 0 rz -90 deg; joints [-13.658, -75.714, -98.895, -5.391, 103.658, -90]
  MoveL 238 to (-678.85, -219.76, 873) mm, rotated rx 180 ry 0 rz -90 deg; joints [-15.07, -75.21, -100.993, -3.797, 105.07, -90]
  MoveL 239 to (-682.74, -207.25, 878) mm, rotated rx 180 ry 0 rz -90 deg; joints [-16.104, -74.873, -103.064, -2.063, 106.104, -90]
  MoveL 240 to (-682.74, -193.48, 878) mm, rotated rx 180 ry 0 rz -90 deg; joints [-16.104, -74.838, -105.1, -0.062, 106.104, -90]
  MoveL 241 to (-685.07, -180.33, 881) mm, rotated rx 180 ry 0 rz -90 deg; joints [-16.733, -74.723, -107.103, 1.826, 106.733, -90]
  MoveL 242 to (-685.07, -166.51, 881) mm, rotated rx 180 ry 0 rz -90 deg; joints [-16.733, -74.821, -109.053, 3.873, 106.733, -90]
  MoveL 243 to (-689.74, -153.73, 887) mm, rotated rx 180 ry 0 rz -90 deg; joints [-18.014, -74.703, -111.009, 5.712, 108.014, -90]
  MoveL 244 to (-687.41, -139.35, 884) mm, rotated rx 180 ry 0 rz -90 deg; joints [-17.37, -75.084, -112.851, 7.935, 107.37, -90]
  MoveL 245 to (-685.85, -125.21, 882) mm, rotated rx 180 ry 0 rz -90 deg; joints [-16.945, -75.505, -114.639, 10.144, 106.945, -90]
  MoveL 246 to (-679.63, -110.37, 874) mm, rotated rx 180 ry 0 rz -90 deg; joints [-15.275, -76.349, -116.232, 12.581, 105.275, -90]
  MoveL 247 to (-678.07, -96.44, 872) mm, rotated rx 180 ry 0 rz -90 deg; joints [-14.866, -76.959, -117.872, 14.831, 104.866, -90]
  MoveL 248 to (-673.41, -82.2, 866) mm, rotated rx 180 ry 0 rz -90 deg; joints [-13.658, -77.912, -119.316, 17.228, 103.658, -90]
  MoveL 249 to (-680.41, -69.33, 875) mm, rotated rx 180 ry 0 rz -90 deg; joints [-15.481, -78.024, -121.209, 19.233, 105.481, -90]
  MoveL 250 to (-663.3, -54.21, 853) mm, rotated rx 180 ry 0 rz -90 deg; joints [-11.145, -80.233, -121.841, 22.075, 101.145, -90]
  MoveL 251 to (-661.74, -40.74, 851) mm, rotated rx 180 ry 0 rz -90 deg; joints [-10.771, -81.223, -123.18, 24.403, 100.771, -90]
  MoveL 252 to (-663.3, -27.46, 853) mm, rotated rx 180 ry 0 rz -90 deg; joints [-11.145, -82.014, -124.677, 26.691, 101.145, -90]
  MoveL 253 to (-652.41, -13.85, 839) mm, rotated rx 180 ry 0 rz -90 deg; joints [-8.596, -84.091, -125.157, 29.249, 98.596, -90]
  MoveL 254 to (-650.08, -0.69, 836) mm, rotated rx 180 ry 0 rz -90 deg; joints [-8.071, -85.431, -126.2, 31.631, 98.071, -90]
  MoveL 255 to (-648.53, 12.39, 834) mm, rotated rx 180 ry 0 rz -90 deg; joints [-7.726, -86.781, -127.241, 34.022, 97.726, -90]
  MoveL 256 to (-642.3, 25.22, 826) mm, rotated rx 180 ry 0 rz -90 deg; joints [-6.376, -88.678, -127.737, 36.415, 96.376, -90]
  MoveL 257 to (-639.97, 38.04, 823) mm, rotated rx 180 ry 0 rz -90 deg; joints [-5.883, -90.262, -128.535, 38.797, 95.883, -90]
  MoveL 258 to (-631.42, 50.26, 812) mm, rotated rx 180 ry 0 rz -90 deg; joints [-4.137, -92.525, -128.522, 41.047, 94.137, -90]
  MoveL 259 to (-629.09, 62.76, 809) mm, rotated rx 180 ry 0 rz -90 deg; joints [-3.678, -94.23, -129.134, 43.364, 93.678, -90]
  MoveL 260 to (-622.86, 74.7, 801) mm, rotated rx 180 ry 0 rz -90 deg; joints [-2.486, -96.352, -129.157, 45.509, 92.486, -90]
  MoveL 261 to (-615.87, 86.28, 792) mm, rotated rx 180 ry 0 rz -90 deg; joints [-1.202, -98.566, -128.947, 47.513, 91.202, -90]
  MoveL 262 to (-618.98, 99.2, 796) mm, rotated rx 180 ry 0 rz -90 deg; joints [-1.766, -99.936, -130.077, 50.013, 91.766, -90]
  MoveL 263 to (-614.31, 110.84, 790) mm, rotated rx 180 ry 0 rz -90 deg; joints [-0.925, -102.005, -130.032, 52.037, 90.925, -90]
  MoveL 264 to (-609.64, 122.3, 784) mm, rotated rx 180 ry 0 rz -90 deg; joints [-0.111, -104.081, -129.892, 53.973, 90.111, -90]
  MoveL 265 to (-638.49, -486.91, 838) mm, rotated rx 180 ry 0 rz -90 deg; joints [-5.896, -92.318, -42.285, -45.397, 95.896, -90]
  MoveL 266 to (-637.73, -473.2, 837) mm, rotated rx 180 ry 0 rz -90 deg; joints [-5.728, -90.572, -46.878, -42.55, 95.728, -90]
  MoveL 267 to (-633.92, -457.33, 832) mm, rotated rx 180 ry 0 rz -90 deg; joints [-4.901, -89.126, -51.391, -39.484, 94.901, -90]
  MoveL 268 to (-632.4, -443.21, 830) mm, rotated rx 180 ry 0 rz -90 deg; joints [-4.576, -87.824, -55.267, -36.909, 94.576, -90]
  MoveL 269 to (-633.16, -430.72, 831) mm, rotated rx 180 ry 0 rz -90 deg; joints [-4.738, -86.566, -58.694, -34.74, 94.738, -90]
  MoveL 270 to (-632.4, -417.18, 830) mm, rotated rx 180 ry 0 rz -90 deg; joints [-4.576, -85.485, -62.049, -32.465, 94.576, -90]
  MoveL 271 to (-641.54, -410.01, 842) mm, rotated rx 180 ry 0 rz -90 deg; joints [-6.577, -83.985, -64.608, -31.407, 96.577, -90]
  MoveL 272 to (-639.26, -395.39, 839) mm, rotated rx 180 ry 0 rz -90 deg; joints [-6.065, -83.124, -67.818, -29.058, 96.065, -90]
  MoveL 273 to (-634.69, -379.5, 833) mm, rotated rx 180 ry 0 rz -90 deg; joints [-5.065, -82.519, -70.953, -26.528, 95.065, -90]
  MoveL 274 to (-635.45, -366.88, 834) mm, rotated rx 180 ry 0 rz -90 deg; joints [-5.229, -81.669, -73.706, -24.625, 95.229, -90]
  MoveL 275 to (-636.97, -354.65, 836) mm, rotated rx 180 ry 0 rz -90 deg; joints [-5.561, -80.827, -76.347, -22.826, 95.561, -90]
  MoveL 276 to (-633.92, -339.91, 832) mm, rotated rx 180 ry 0 rz -90 deg; joints [-4.901, -80.389, -79.019, -20.592, 94.901, -90]
  MoveL 277 to (-641.54, -330.79, 842) mm, rotated rx 180 ry 0 rz -90 deg; joints [-6.577, -79.19, -81.389, -19.42, 96.577, -90]
  MoveL 278 to (-642.3, -317.96, 843) mm, rotated rx 180 ry 0 rz -90 deg; joints [-6.749, -78.563, -83.854, -17.584, 96.749, -90]
  MoveL 279 to (-640.78, -304.02, 841) mm, rotated rx 180 ry 0 rz -90 deg; joints [-6.405, -78.175, -86.277, -15.548, 96.405, -90]
  MoveL 280 to (-640.02, -290.48, 840) mm, rotated rx 180 ry 0 rz -90 deg; joints [-6.235, -77.792, -88.613, -13.596, 96.235, -90]
  MoveL 281 to (-649.92, -281.6, 853) mm, rotated rx 180 ry 0 rz -90 deg; joints [-8.522, -76.566, -90.867, -12.567, 98.522, -90]
  MoveL 282 to (-645.35, -266.34, 847) mm, rotated rx 180 ry 0 rz -90 deg; joints [-7.448, -76.59, -93.123, -10.287, 97.448, -90]
  MoveL 283 to (-657.54, -257.84, 863) mm, rotated rx 180 ry 0 rz -90 deg; joints [-10.384, -75.283, -95.34, -9.376, 100.384, -90]
  MoveL 284 to (-653.73, -242.89, 858) mm, rotated rx 180 ry 0 rz -90 deg; joints [-9.442, -75.324, -97.516, -7.159, 99.442, -90]
  MoveL 285 to (-662.11, -232.38, 869) mm, rotated rx 180 ry 0 rz -90 deg; joints [-11.545, -74.445, -99.691, -5.864, 101.545, -90]
  MoveL 286 to (-668.21, -220.76, 877) mm, rotated rx 180 ry 0 rz -90 deg; joints [-13.144, -73.829, -101.826, -4.345, 103.144, -90]
  MoveL 287 to (-664.4, -205.83, 872) mm, rotated rx 180 ry 0 rz -90 deg; joints [-12.138, -74.007, -103.885, -2.108, 102.138, -90]
  MoveL 288 to (-668.97, -193.48, 878) mm, rotated rx 180 ry 0 rz -90 deg; joints [-13.348, -73.614, -105.963, -0.422, 103.348, -90]
  MoveL 289 to (-672.02, -180.53, 882) mm, rotated rx 180 ry 0 rz -90 deg; joints [-14.173, -73.406, -107.999, 1.404, 104.173, -90]
  MoveL 290 to (-671.26, -166.51, 881) mm, rotated rx 180 ry 0 rz -90 deg; joints [-13.965, -73.547, -109.95, 3.497, 103.965, -90]
  MoveL 291 to (-670.5, -152.52, 880) mm, rotated rx 180 ry 0 rz -90 deg; joints [-13.759, -73.764, -111.848, 5.612, 103.759, -90]
  MoveL 292 to (-671.26, -138.88, 881) mm, rotated rx 180 ry 0 rz -90 deg; joints [-13.965, -73.937, -113.733, 7.67, 103.965, -90]
  MoveL 293 to (-664.4, -123.79, 872) mm, rotated rx 180 ry 0 rz -90 deg; joints [-12.138, -74.832, -115.333, 10.165, 102.138, -90]
  MoveL 294 to (-666.69, -110.49, 875) mm, rotated rx 180 ry 0 rz -90 deg; joints [-12.739, -75.029, -117.171, 12.2, 102.739, -90]
  MoveL 295 to (-662.88, -96.22, 870) mm, rotated rx 180 ry 0 rz -90 deg; joints [-11.742, -75.857, -118.717, 14.574, 101.742, -90]
  MoveL 296 to (-658.3, -82.01, 864) mm, rotated rx 180 ry 0 rz -90 deg; joints [-10.575, -76.87, -120.13, 17, 100.575, -90]
  MoveL 297 to (-659.07, -68.54, 865) mm, rotated rx 180 ry 0 rz -90 deg; joints [-10.768, -77.457, -121.76, 19.217, 100.768, -90]
  MoveL 298 to (-653.73, -54.53, 858) mm, rotated rx 180 ry 0 rz -90 deg; joints [-9.442, -78.752, -122.957, 21.709, 99.442, -90]
  MoveL 299 to (-649.92, -40.83, 853) mm, rotated rx 180 ry 0 rz -90 deg; joints [-8.522, -80.002, -124.15, 24.151, 98.522, -90]
  MoveL 300 to (-648.4, -27.39, 851) mm, rotated rx 180 ry 0 rz -90 deg; joints [-8.16, -81.105, -125.435, 26.54, 98.16, -90]
  MoveL 301 to (-640.02, -13.87, 840) mm, rotated rx 180 ry 0 rz -90 deg; joints [-6.235, -83.064, -126.039, 29.103, 96.235, -90]
  MoveL 302 to (-640.02, -0.69, 840) mm, rotated rx 180 ry 0 rz -90 deg; joints [-6.235, -84.181, -127.305, 31.487, 96.235, -90]
  MoveL 303 to (-632.4, 12.33, 830) mm, rotated rx 180 ry 0 rz -90 deg; joints [-4.576, -86.248, -127.721, 33.969, 94.576, -90]
  MoveL 304 to (-627.83, 25.16, 824) mm, rotated rx 180 ry 0 rz -90 deg; joints [-3.622, -88.051, -128.329, 36.38, 93.622, -90]
  MoveL 305 to (-620.21, 37.62, 814) mm, rotated rx 180 ry 0 rz -90 deg; joints [-2.098, -90.272, -128.448, 38.719, 92.098, -90]
  MoveL 306 to (-623.26, 50.63, 818) mm, rotated rx 180 ry 0 rz -90 deg; joints [-2.698, -91.36, -129.815, 41.176, 92.698, -90]
  MoveL 307 to (-614.11, 62.53, 806) mm, rotated rx 180 ry 0 rz -90 deg; joints [-0.936, -93.844, -129.513, 43.358, 90.937, -90]
  MoveL 308 to (-608.02, 74.42, 798) mm, rotated rx 180 ry 0 rz -90 deg; joints [0.176, -96.028, -129.476, 45.505, 89.824, -90]
  MoveL 309 to (-604.21, 86.39, 793) mm, rotated rx 180 ry 0 rz -90 deg; joints [0.847, -98, -129.667, 47.668, 89.153, -90]
  MoveL 310 to (-606.49, 99.2, 796) mm, rotated rx 180 ry 0 rz -90 deg; joints [0.446, -99.442, -130.712, 50.154, 89.554, -90]
  MoveL 311 to (-599.64, 110.42, 787) mm, rotated rx 180 ry 0 rz -90 deg; joints [1.628, -101.755, -130.273, 52.028, 88.372, -90]
  MoveL 312 to (-601.16, 123.08, 789) mm, rotated rx 180 ry 0 rz -90 deg; joints [1.37, -103.392, -131.078, 54.471, 88.63, -90]
  MoveL 313 to (-623.86, -485.75, 836) mm, rotated rx 180 ry 0 rz -90 deg; joints [-2.987, -91.501, -43.384, -45.114, 92.987, -90]
  MoveL 314 to (-626.1, -474.33, 839) mm, rotated rx 180 ry 0 rz -90 deg; joints [-3.466, -89.736, -47.493, -42.771, 93.466, -90]
  MoveL 315 to (-623.86, -459.53, 836) mm, rotated rx 180 ry 0 rz -90 deg; joints [-2.987, -88.266, -51.806, -39.928, 92.987, -90]
  MoveL 316 to (-620.88, -444.28, 832) mm, rotated rx 180 ry 0 rz -90 deg; joints [-2.36, -87.027, -55.82, -37.153, 92.36, -90]
  MoveL 317 to (-622.37, -432.27, 834) mm, rotated rx 180 ry 0 rz -90 deg; joints [-2.671, -85.722, -59.186, -35.092, 92.671, -90]
  MoveL 318 to (-620.88, -418.19, 832) mm, rotated rx 180 ry 0 rz -90 deg; joints [-2.36, -84.681, -62.591, -32.728, 92.36, -90]
  MoveL 319 to (-622.37, -406.11, 834) mm, rotated rx 180 ry 0 rz -90 deg; joints [-2.671, -83.558, -65.64, -30.801, 92.671, -90]
  MoveL 320 to (-621.62, -392.56, 833) mm, rotated rx 180 ry 0 rz -90 deg; joints [-2.515, -82.66, -68.682, -28.657, 92.515, -90]
  MoveL 321 to (-617.15, -376.77, 827) mm, rotated rx 180 ry 0 rz -90 deg; joints [-1.595, -82.138, -71.718, -26.144, 91.595, -90]
  MoveL 322 to (-620.88, -366, 832) mm, rotated rx 180 ry 0 rz -90 deg; joints [-2.36, -81.053, -74.353, -24.594, 92.36, -90]
  MoveL 323 to (-618.64, -351.68, 829) mm, rotated rx 180 ry 0 rz -90 deg; joints [-1.898, -80.519, -77.066, -22.415, 91.898, -90]
  MoveL 324 to (-623.86, -341.54, 836) mm, rotated rx 180 ry 0 rz -90 deg; joints [-2.987, -79.401, -79.551, -21.048, 92.987, -90]
  MoveL 325 to (-622.37, -327.64, 834) mm, rotated rx 180 ry 0 rz -90 deg; joints [-2.671, -78.921, -82.086, -18.993, 92.671, -90]
  MoveL 326 to (-626.1, -316.45, 839) mm, rotated rx 180 ry 0 rz -90 deg; joints [-3.466, -78.022, -84.5, -17.477, 93.467, -90]
  MoveL 327 to (-625.35, -302.93, 838) mm, rotated rx 180 ry 0 rz -90 deg; joints [-3.306, -77.587, -86.89, -15.522, 93.306, -90]
  MoveL 328 to (-627.59, -290.83, 841) mm, rotated rx 180 ry 0 rz -90 deg; joints [-3.791, -76.921, -89.219, -13.86, 93.791, -90]
  MoveL 329 to (-627.59, -277.64, 841) mm, rotated rx 180 ry 0 rz -90 deg; joints [-3.791, -76.524, -91.491, -11.986, 93.791, -90]
  MoveL 330 to (-632.82, -266.66, 848) mm, rotated rx 180 ry 0 rz -90 deg; joints [-4.955, -75.655, -93.764, -10.581, 94.955, -90]
  MoveL 331 to (-646.25, -258.74, 866) mm, rotated rx 180 ry 0 rz -90 deg; joints [-8.16, -74.1, -96.048, -9.852, 98.16, -90]
  MoveL 332 to (-644.01, -244.31, 863) mm, rotated rx 180 ry 0 rz -90 deg; joints [-7.604, -74.016, -98.239, -7.746, 97.604, -90]
  MoveL 333 to (-649.98, -232.91, 871) mm, rotated rx 180 ry 0 rz -90 deg; joints [-9.106, -73.257, -100.44, -6.303, 99.106, -90]
  MoveL 334 to (-649.98, -219.25, 871) mm, rotated rx 180 ry 0 rz -90 deg; joints [-9.106, -73.082, -102.563, -4.355, 99.106, -90]
  MoveL 335 to (-649.23, -205.36, 870) mm, rotated rx 180 ry 0 rz -90 deg; joints [-8.915, -73.04, -104.624, -2.336, 98.915, -90]
  MoveL 336 to (-646.99, -191.06, 867) mm, rotated rx 180 ry 0 rz -90 deg; joints [-8.347, -73.213, -106.595, -0.193, 98.347, -90]
  MoveL 337 to (-649.23, -178.07, 870) mm, rotated rx 180 ry 0 rz -90 deg; joints [-8.915, -73.017, -108.624, 1.641, 98.915, -90]
  MoveL 338 to (-650.73, -164.81, 872) mm, rotated rx 180 ry 0 rz -90 deg; joints [-9.298, -72.959, -110.603, 3.562, 99.298, -90]
  MoveL 339 to (-654.46, -152, 877) mm, rotated rx 180 ry 0 rz -90 deg; joints [-10.274, -72.751, -112.62, 5.371, 100.274, -90]
  MoveL 340 to (-644.01, -136.04, 863) mm, rotated rx 180 ry 0 rz -90 deg; joints [-7.604, -74.066, -114.061, 8.127, 97.604, -90]
  MoveL 341 to (-649.23, -123.5, 870) mm, rotated rx 180 ry 0 rz -90 deg; joints [-8.915, -73.817, -116.088, 9.905, 98.915, -90]
  MoveL 342 to (-644.01, -108.98, 863) mm, rotated rx 180 ry 0 rz -90 deg; joints [-7.604, -74.787, -117.57, 12.357, 97.604, -90]
  MoveL 343 to (-644.01, -95.44, 863) mm, rotated rx 180 ry 0 rz -90 deg; joints [-7.604, -75.269, -119.258, 14.527, 97.604, -90]
  MoveL 344 to (-638.79, -81.25, 856) mm, rotated rx 180 ry 0 rz -90 deg; joints [-6.341, -76.455, -120.552, 17.007, 96.341, -90]
  MoveL 345 to (-640.28, -67.98, 858) mm, rotated rx 180 ry 0 rz -90 deg; joints [-6.697, -76.934, -122.236, 19.17, 96.697, -90]
  MoveL 346 to (-639.53, -54.46, 857) mm, rotated rx 180 ry 0 rz -90 deg; joints [-6.519, -77.774, -123.713, 21.488, 96.519, -90]
  MoveL 347 to (-644.01, -41.31, 863) mm, rotated rx 180 ry 0 rz -90 deg; joints [-7.604, -78.096, -125.55, 23.646, 97.604, -90]
  MoveL 348 to (-634.31, -27.36, 850) mm, rotated rx 180 ry 0 rz -90 deg; joints [-5.296, -80.198, -126.169, 26.367, 95.296, -90]
  MoveL 349 to (-625.35, -13.83, 838) mm, rotated rx 180 ry 0 rz -90 deg; joints [-3.306, -82.365, -126.634, 28.999, 93.306, -90]
  MoveL 350 to (-626.1, -0.69, 839) mm, rotated rx 180 ry 0 rz -90 deg; joints [-3.467, -83.39, -127.988, 31.378, 93.467, -90]
  MoveL 351 to (-624.61, 12.43, 837) mm, rotated rx 180 ry 0 rz -90 deg; joints [-3.146, -84.798, -129.042, 33.84, 93.146, -90]
  MoveL 352 to (-615.65, 25.19, 825) mm, rotated rx 180 ry 0 rz -90 deg; joints [-1.295, -87.226, -129.114, 36.34, 91.295, -90]
  MoveL 353 to (-608.94, 37.71, 816) mm, rotated rx 180 ry 0 rz -90 deg; joints [0.012, -89.441, -129.292, 38.734, 89.988, -90]
  MoveL 354 to (-607.44, 50.39, 814) mm, rotated rx 180 ry 0 rz -90 deg; joints [0.293, -91.064, -130.073, 41.137, 89.707, -90]
  MoveL 355 to (-599.98, 62.38, 804) mm, rotated rx 180 ry 0 rz -90 deg; joints [1.653, -93.464, -129.899, 43.363, 88.347, -90]
  MoveL 356 to (-594.76, 74.33, 797) mm, rotated rx 180 ry 0 rz -90 deg; joints [2.56, -95.621, -129.928, 45.549, 87.44, -90]
  MoveL 357 to (-592.52, 86.5, 794) mm, rotated rx 180 ry 0 rz -90 deg; joints [2.937, -97.471, -130.335, 47.806, 87.063, -90]
  MoveL 358 to (-589.53, 98.45, 790) mm, rotated rx 180 ry 0 rz -90 deg; joints [3.43, -99.442, -130.542, 49.983, 86.57, -90]
  MoveL 359 to (-588.79, 110.7, 789) mm, rotated rx 180 ry 0 rz -90 deg; joints [3.552, -101.231, -131.048, 52.279, 86.448, -90]
  MoveL 360 to (-591.03, 123.54, 792) mm, rotated rx 180 ry 0 rz -90 deg; joints [3.185, -102.831, -131.996, 54.827, 86.815, -90]
  MoveL 361 to (-612.94, -487.49, 839) mm, rotated rx 180 ry 0 rz -90 deg; joints [-0.808, -90.711, -43.836, -45.453, 90.808, -90]
  MoveL 362 to (-606.37, -469.24, 830) mm, rotated rx 180 ry 0 rz -90 deg; joints [0.524, -89.238, -48.988, -41.774, 89.476, -90]
  MoveL 363 to (-609.29, -458.43, 834) mm, rotated rx 180 ry 0 rz -90 deg; joints [-0.059, -87.627, -52.621, -39.752, 90.059, -90]
  MoveL 364 to (-612.94, -448.02, 839) mm, rotated rx 180 ry 0 rz -90 deg; joints [-0.808, -86.085, -55.997, -37.918, 90.808, -90]
  MoveL 365 to (-607.83, -431.23, 832) mm, rotated rx 180 ry 0 rz -90 deg; joints [0.235, -85.138, -59.893, -34.969, 89.766, -90]
  MoveL 366 to (-609.29, -419.19, 834) mm, rotated rx 180 ry 0 rz -90 deg; joints [-0.059, -83.921, -63.079, -33, 90.059, -90]
  MoveL 367 to (-607.83, -405.14, 832) mm, rotated rx 180 ry 0 rz -90 deg; joints [0.235, -82.998, -66.284, -30.719, 89.766, -90]
  MoveL 368 to (-601.25, -387.85, 823) mm, rotated rx 180 ry 0 rz -90 deg; joints [1.511, -82.613, -69.503, -27.884, 88.489, -90]
  MoveL 369 to (-606.37, -378.14, 830) mm, rotated rx 180 ry 0 rz -90 deg; joints [0.524, -81.318, -72.173, -26.509, 89.476, -90]
  MoveL 370 to (-605.64, -364.68, 829) mm, rotated rx 180 ry 0 rz -90 deg; joints [0.668, -80.597, -74.934, -24.469, 89.332, -90]
  MoveL 371 to (-605.64, -351.68, 829) mm, rotated rx 180 ry 0 rz -90 deg; joints [0.668, -79.877, -77.58, -22.543, 89.332, -90]
  MoveL 372 to (-610.75, -341.54, 836) mm, rotated rx 180 ry 0 rz -90 deg; joints [-0.356, -78.712, -80.088, -21.2, 90.356, -90]
  MoveL 373 to (-611.48, -328.82, 837) mm, rotated rx 180 ry 0 rz -90 deg; joints [-0.505, -78.02, -82.598, -19.382, 90.506, -90]
  MoveL 374 to (-611.48, -315.7, 837) mm, rotated rx 180 ry 0 rz -90 deg; joints [-0.505, -77.457, -85.045, -17.498, 90.506, -90]
  MoveL 375 to (-612.94, -303.3, 839) mm, rotated rx 180 ry 0 rz -90 deg; joints [-0.808, -76.795, -87.43, -15.775, 90.808, -90]
  MoveL 376 to (-618.06, -292.56, 846) mm, rotated rx 180 ry 0 rz -90 deg; joints [-1.895, -75.792, -89.79, -14.418, 91.895, -90]
  MoveL 377 to (-610.02, -275.66, 835) mm, rotated rx 180 ry 0 rz -90 deg; joints [-0.207, -76.279, -91.967, -11.754, 90.207, -90]
  MoveL 378 to (-614.4, -264.45, 841) mm, rotated rx 180 ry 0 rz -90 deg; joints [-1.114, -75.43, -94.254, -10.316, 91.114, -90]
  MoveL 379 to (-632.67, -258.74, 866) mm, rotated rx 180 ry 0 rz -90 deg; joints [-5.262, -73.151, -96.703, -10.146, 95.262, -90]
  MoveL 380 to (-630.48, -244.31, 863) mm, rotated rx 180 ry 0 rz -90 deg; joints [-4.731, -73.081, -98.884, -8.035, 94.731, -90]
  MoveL 381 to (-634.86, -232.38, 869) mm, rotated rx 180 ry 0 rz -90 deg; joints [-5.802, -72.394, -101.104, -6.502, 95.802, -90]
  MoveL 382 to (-641.44, -221.02, 878) mm, rotated rx 180 ry 0 rz -90 deg; joints [-7.478, -71.551, -103.331, -5.119, 97.478, -90]
  MoveL 383 to (-632.67, -204.42, 866) mm, rotated rx 180 ry 0 rz -90 deg; joints [-5.262, -72.334, -105.24, -2.426, 95.262, -90]
  MoveL 384 to (-632.67, -190.84, 866) mm, rotated rx 180 ry 0 rz -90 deg; joints [-5.262, -72.286, -107.256, -0.458, 95.262, -90]
  MoveL 385 to (-638.51, -178.89, 874) mm, rotated rx 180 ry 0 rz -90 deg; joints [-6.722, -71.646, -109.425, 1.071, 96.722, -90]
  MoveL 386 to (-637.05, -164.81, 872) mm, rotated rx 180 ry 0 rz -90 deg; joints [-6.351, -71.882, -111.327, 3.209, 96.351, -90]
  MoveL 387 to (-635.59, -150.79, 870) mm, rotated rx 180 ry 0 rz -90 deg; joints [-5.984, -72.199, -113.169, 5.368, 95.984, -90]
  MoveL 388 to (-638.51, -137.78, 874) mm, rotated rx 180 ry 0 rz -90 deg; joints [-6.722, -72.08, -115.159, 7.24, 96.722, -90]
  MoveL 389 to (-629.75, -122.37, 862) mm, rotated rx 180 ry 0 rz -90 deg; joints [-4.557, -73.457, -116.505, 9.962, 94.557, -90]
  MoveL 390 to (-635.59, -109.86, 870) mm, rotated rx 180 ry 0 rz -90 deg; joints [-5.984, -73.11, -118.601, 11.711, 95.984, -90]
  MoveL 391 to (-631.94, -95.66, 865) mm, rotated rx 180 ry 0 rz -90 deg; joints [-5.084, -74.04, -120.09, 14.13, 95.084, -90]
  MoveL 392 to (-629.02, -81.72, 861) mm, rotated rx 180 ry 0 rz -90 deg; joints [-4.383, -74.984, -121.541, 16.524, 94.383, -90]
  MoveL 393 to (-623.9, -67.66, 854) mm, rotated rx 180 ry 0 rz -90 deg; joints [-3.194, -76.332, -122.727, 19.06, 93.194, -90]
  MoveL 394 to (-621.71, -54.08, 851) mm, rotated rx 180 ry 0 rz -90 deg; joints [-2.7, -77.386, -124.064, 21.45, 92.7, -90]
  MoveL 395 to (-625.36, -40.98, 856) mm, rotated rx 180 ry 0 rz -90 deg; joints [-3.529, -77.723, -125.884, 23.607, 93.529, -90]
  MoveL 396 to (-619.52, -27.3, 848) mm, rotated rx 180 ry 0 rz -90 deg; joints [-2.214, -79.476, -126.747, 26.223, 92.214, -90]
  MoveL 397 to (-610.75, -13.8, 836) mm, rotated rx 180 ry 0 rz -90 deg; joints [-0.356, -81.766, -127.136, 28.902, 90.356, -90]
  MoveL 398 to (-610.75, -0.69, 836) mm, rotated rx 180 ry 0 rz -90 deg; joints [-0.356, -82.887, -128.415, 31.302, 90.356, -90]
  MoveL 399 to (-610.02, 12.4, 835) mm, rotated rx 180 ry 0 rz -90 deg; joints [-0.207, -84.213, -129.549, 33.761, 90.207, -90]
  MoveL 400 to (-606.37, 25.35, 830) mm, rotated rx 180 ry 0 rz -90 deg; joints [0.524, -86.039, -130.235, 36.274, 89.476, -90]
  MoveL 401 to (-599.06, 37.9, 820) mm, rotated rx 180 ry 0 rz -90 deg; joints [1.922, -88.44, -130.303, 38.742, 88.079, -90]
  MoveL 402 to (-593.22, 50.26, 812) mm, rotated rx 180 ry 0 rz -90 deg; joints [2.98, -90.689, -130.431, 41.121, 87.02, -90]
  MoveL 403 to (-584.45, 62.07, 800) mm, rotated rx 180 ry 0 rz -90 deg; joints [4.474, -93.357, -129.952, 43.31, 85.526, -90]
  MoveL 404 to (-582.26, 74.33, 797) mm, rotated rx 180 ry 0 rz -90 deg; joints [4.831, -95.187, -130.425, 45.612, 85.169, -90]
  MoveL 405 to (-577.15, 86.07, 790) mm, rotated rx 180 ry 0 rz -90 deg; joints [5.639, -97.414, -130.309, 47.723, 84.362, -90]
  MoveL 406 to (-574.95, 98.08, 787) mm, rotated rx 180 ry 0 rz -90 deg; joints [5.975, -99.316, -130.617, 49.933, 84.026, -90]
  MoveL 407 to (-576.42, 110.7, 789) mm, rotated rx 180 ry 0 rz -90 deg; joints [5.751, -100.882, -131.516, 52.398, 84.249, -90]
  MoveL 408 to (-574.95, 122.76, 787) mm, rotated rx 180 ry 0 rz -90 deg; joints [5.975, -102.816, -131.82, 54.636, 84.026, -90]
  MoveL 409 to (-599.79, -487.49, 839) mm, rotated rx 180 ry 0 rz -90 deg; joints [1.904, -90.028, -44.526, -45.446, 88.096, -90]
  MoveL 410 to (-594.78, -470.37, 832) mm, rotated rx 180 ry 0 rz -90 deg; joints [2.873, -88.561, -49.425, -42.014, 87.127, -90]
  MoveL 411 to (-594.07, -456.78, 831) mm, rotated rx 180 ry 0 rz -90 deg; joints [3.008, -87.132, -53.397, -39.471, 86.992, -90]
  MoveL 412 to (-591.92, -442.15, 828) mm, rotated rx 180 ry 0 rz -90 deg; joints [3.408, -85.953, -57.196, -36.851, 86.592, -90]
  MoveL 413 to (-594.07, -430.72, 831) mm, rotated rx 180 ry 0 rz -90 deg; joints [3.008, -84.596, -60.463, -34.941, 86.992, -90]
  MoveL 414 to (-594.07, -417.68, 831) mm, rotated rx 180 ry 0 rz -90 deg; joints [3.008, -83.488, -63.713, -32.799, 86.992, -90]
  MoveL 415 to (-593.35, -404.17, 830) mm, rotated rx 180 ry 0 rz -90 deg; joints [3.142, -82.532, -66.841, -30.627, 86.858, -90]
  MoveL 416 to (-587.63, -387.38, 822) mm, rotated rx 180 ry 0 rz -90 deg; joints [4.185, -82.148, -69.97, -27.881, 85.815, -90]
  MoveL 417 to (-589.78, -375.86, 825) mm, rotated rx 180 ry 0 rz -90 deg; joints [3.8, -81.098, -72.724, -26.179, 86.2, -90]
  MoveL 418 to (-592.64, -364.68, 829) mm, rotated rx 180 ry 0 rz -90 deg; joints [3.276, -80.024, -75.392, -24.583, 86.724, -90]
  MoveL 419 to (-595.5, -353.38, 833) mm, rotated rx 180 ry 0 rz -90 deg; joints [2.737, -78.997, -78.002, -23.001, 87.263, -90]
  MoveL 420 to (-593.35, -339.09, 830) mm, rotated rx 180 ry 0 rz -90 deg; joints [3.142, -78.562, -80.587, -20.851, 86.858, -90]
  MoveL 421 to (-600.5, -330, 840) mm, rotated rx 180 ry 0 rz -90 deg; joints [1.761, -77.153, -83.069, -19.779, 88.239, -90]
  MoveL 422 to (-599.79, -316.45, 839) mm, rotated rx 180 ry 0 rz -90 deg; joints [1.904, -76.658, -85.525, -17.817, 88.096, -90]
  MoveL 423 to (-597.64, -302.21, 836) mm, rotated rx 180 ry 0 rz -90 deg; joints [2.325, -76.397, -87.889, -15.714, 87.675, -90]
  MoveL 424 to (-599.79, -290.14, 839) mm, rotated rx 180 ry 0 rz -90 deg; joints [1.904, -75.682, -90.235, -14.083, 88.096, -90]
  MoveL 425 to (-606.22, -279.95, 848) mm, rotated rx 180 ry 0 rz -90 deg; joints [0.591, -74.491, -92.614, -12.896, 89.409, -90]
  MoveL 426 to (-602.65, -265.08, 843) mm, rotated rx 180 ry 0 rz -90 deg; joints [1.329, -74.564, -94.78, -10.656, 88.671, -90]
  MoveL 427 to (-613.37, -256.35, 858) mm, rotated rx 180 ry 0 rz -90 deg; joints [-0.96, -72.928, -97.208, -9.863, 90.96, -90]
  MoveL 428 to (-617.66, -244.59, 864) mm, rotated rx 180 ry 0 rz -90 deg; joints [-1.939, -72.132, -99.481, -8.387, 91.939, -90]
  MoveL 429 to (-619.09, -231.58, 866) mm, rotated rx 180 ry 0 rz -90 deg; joints [-2.273, -71.721, -101.669, -6.61, 92.273, -90]
  MoveL 430 to (-624.09, -219.76, 873) mm, rotated rx 180 ry 0 rz -90 deg; joints [-3.478, -70.942, -103.911, -5.147, 93.478, -90]
  MoveL 431 to (-619.8, -204.65, 867) mm, rotated rx 180 ry 0 rz -90 deg; joints [-2.442, -71.325, -105.874, -2.801, 92.442, -90]
  MoveL 432 to (-616.23, -189.95, 862) mm, rotated rx 180 ry 0 rz -90 deg; joints [-1.608, -71.728, -107.756, -0.516, 91.608, -90]
  MoveL 433 to (-619.09, -177.26, 866) mm, rotated rx 180 ry 0 rz -90 deg; joints [-2.273, -71.363, -109.85, 1.213, 92.273, -90]
  MoveL 434 to (-623.38, -164.81, 872) mm, rotated rx 180 ry 0 rz -90 deg; joints [-3.303, -70.875, -111.985, 2.86, 93.303, -90]
  MoveL 435 to (-623.38, -151.14, 872) mm, rotated rx 180 ry 0 rz -90 deg; joints [-3.303, -71.011, -113.899, 4.909, 93.303, -90]
  MoveL 436 to (-618.37, -136.36, 865) mm, rotated rx 180 ry 0 rz -90 deg; joints [-2.105, -71.906, -115.484, 7.39, 92.105, -90]
  MoveL 437 to (-620.52, -123.22, 868) mm, rotated rx 180 ry 0 rz -90 deg; joints [-2.612, -71.904, -117.424, 9.328, 92.612, -90]
  MoveL 438 to (-622.66, -109.99, 871) mm, rotated rx 180 ry 0 rz -90 deg; joints [-3.129, -71.98, -119.338, 11.318, 93.129, -90]
  MoveL 439 to (-619.8, -95.89, 867) mm, rotated rx 180 ry 0 rz -90 deg; joints [-2.442, -72.845, -120.872, 13.717, 92.442, -90]
  MoveL 440 to (-613.37, -81.44, 858) mm, rotated rx 180 ry 0 rz -90 deg; joints [-0.96, -74.351, -122.028, 16.379, 90.96, -90]
  MoveL 441 to (-613.37, -67.98, 858) mm, rotated rx 180 ry 0 rz -90 deg; joints [-0.96, -75, -123.633, 18.633, 90.96, -90]
  MoveL 442 to (-607.65, -54.02, 850) mm, rotated rx 180 ry 0 rz -90 deg; joints [0.289, -76.632, -124.631, 21.263, 89.711, -90]
  MoveL 443 to (-611.94, -40.98, 856) mm, rotated rx 180 ry 0 rz -90 deg; joints [-0.642, -76.806, -126.562, 23.368, 90.642, -90]
  MoveL 444 to (-605.51, -27.26, 847) mm, rotated rx 180 ry 0 rz -90 deg; joints [0.74, -78.751, -127.313, 26.063, 89.26, -90]
  MoveL 445 to (-596.21, -13.77, 834) mm, rotated rx 180 ry 0 rz -90 deg; joints [2.6, -81.272, -127.545, 28.818, 87.4, -90]
  MoveL 446 to (-601.22, -0.69, 841) mm, rotated rx 180 ry 0 rz -90 deg; joints [1.618, -81.604, -129.478, 31.082, 88.382, -90]
  MoveL 447 to (-592.64, 12.32, 829) mm, rotated rx 180 ry 0 rz -90 deg; joints [3.276, -84.181, -129.561, 33.742, 86.724, -90]
  MoveL 448 to (-590.49, 25.22, 826) mm, rotated rx 180 ry 0 rz -90 deg; joints [3.67, -85.825, -130.406, 36.231, 86.33, -90]
  MoveL 449 to (-586.2, 37.9, 820) mm, rotated rx 180 ry 0 rz -90 deg; joints [4.437, -87.876, -130.841, 38.717, 85.563, -90]
  MoveL 450 to (-578.34, 50.08, 809) mm, rotated rx 180 ry 0 rz -90 deg; joints [5.768, -90.51, -130.577, 41.088, 84.232, -90]
  MoveL 451 to (-574.05, 62.3, 803) mm, rotated rx 180 ry 0 rz -90 deg; joints [6.456, -92.644, -130.768, 43.412, 83.544, -90]
  MoveL 452 to (-571.91, 74.61, 800) mm, rotated rx 180 ry 0 rz -90 deg; joints [6.79, -94.518, -131.241, 45.758, 83.21, -90]
  MoveL 453 to (-564.04, 85.96, 789) mm, rotated rx 180 ry 0 rz -90 deg; joints [7.962, -97.176, -130.572, 47.748, 82.038, -90]
  MoveL 454 to (-564.04, 98.33, 789) mm, rotated rx 180 ry 0 rz -90 deg; joints [7.962, -98.841, -131.275, 50.116, 82.038, -90]
  MoveL 455 to (-562.61, 110.42, 787) mm, rotated rx 180 ry 0 rz -90 deg; joints [8.167, -100.739, -131.639, 52.378, 81.833, -90]
  MoveL 456 to (-560.47, 122.3, 784) mm, rotated rx 180 ry 0 rz -90 deg; joints [8.469, -102.753, -131.792, 54.544, 81.531, -90]
  MoveL 457 to (-584.53, -485.75, 836) mm, rotated rx 180 ry 0 rz -90 deg; joints [5.044, -89.516, -45.397, -45.087, 84.956, -90]
  MoveL 458 to (-581.74, -470.37, 832) mm, rotated rx 180 ry 0 rz -90 deg; joints [5.547, -88.018, -49.944, -42.038, 84.453, -90]
  MoveL 459 to (-582.43, -457.88, 833) mm, rotated rx 180 ry 0 rz -90 deg; joints [5.423, -86.509, -53.763, -39.728, 84.577, -90]
  MoveL 460 to (-575.44, -439.48, 823) mm, rotated rx 180 ry 0 rz -90 deg; joints [6.63, -85.736, -57.877, -36.387, 83.37, -90]
  MoveL 461 to (-580.34, -430.2, 830) mm, rotated rx 180 ry 0 rz -90 deg; joints [5.794, -84.139, -60.954, -34.908, 84.206, -90]
  MoveL 462 to (-578.94, -416.18, 828) mm, rotated rx 180 ry 0 rz -90 deg; joints [6.037, -83.167, -64.248, -32.586, 83.963, -90]
  MoveL 463 to (-578.24, -402.71, 827) mm, rotated rx 180 ry 0 rz -90 deg; joints [6.157, -82.232, -67.339, -30.429, 83.843, -90]
  MoveL 464 to (-575.44, -387.85, 823) mm, rotated rx 180 ry 0 rz -90 deg; joints [6.63, -81.61, -70.337, -28.052, 83.37, -90]
  MoveL 465 to (-574.74, -374.49, 822) mm, rotated rx 180 ry 0 rz -90 deg; joints [6.747, -80.856, -73.142, -26.002, 83.254, -90]
  MoveL 466 to (-581.74, -366, 832) mm, rotated rx 180 ry 0 rz -90 deg; joints [5.547, -79.283, -75.763, -24.954, 84.453, -90]
  MoveL 467 to (-586.63, -355.92, 839) mm, rotated rx 180 ry 0 rz -90 deg; joints [4.658, -77.989, -78.368, -23.643, 85.342, -90]
  MoveL 468 to (-580.34, -339.09, 830) mm, rotated rx 180 ry 0 rz -90 deg; joints [5.794, -78.048, -80.98, -20.972, 84.206, -90]
  MoveL 469 to (-584.53, -328.43, 836) mm, rotated rx 180 ry 0 rz -90 deg; joints [5.044, -76.914, -83.489, -19.596, 84.956, -90]
  MoveL 470 to (-585.93, -316.08, 838) mm, rotated rx 180 ry 0 rz -90 deg; joints [4.787, -76.169, -85.942, -17.89, 85.213, -90]
  MoveL 471 to (-590.13, -305.1, 844) mm, rotated rx 180 ry 0 rz -90 deg; joints [3.996, -75.112, -88.378, -16.51, 86.004, -90]
  MoveL 472 to (-586.63, -290.14, 839) mm, rotated rx 180 ry 0 rz -90 deg; joints [4.658, -75.096, -90.656, -14.249, 85.342, -90]
  MoveL 473 to (-592.22, -279.62, 847) mm, rotated rx 180 ry 0 rz -90 deg; joints [3.587, -73.929, -93.055, -13.016, 86.413, -90]
  MoveL 474 to (-591.52, -266.03, 846) mm, rotated rx 180 ry 0 rz -90 deg; joints [3.724, -73.649, -95.278, -11.072, 86.276, -90]
  MoveL 475 to (-590.13, -252.16, 844) mm, rotated rx 180 ry 0 rz -90 deg; joints [3.996, -73.531, -97.416, -9.053, 86.004, -90]
  MoveL 476 to (-596.42, -241.48, 853) mm, rotated rx 180 ry 0 rz -90 deg; joints [2.745, -72.376, -99.777, -7.847, 87.255, -90]
  MoveL 477 to (-602.01, -230.24, 861) mm, rotated rx 180 ry 0 rz -90 deg; joints [1.566, -71.371, -102.095, -6.534, 88.434, -90]
  MoveL 478 to (-610.4, -219.76, 873) mm, rotated rx 180 ry 0 rz -90 deg; joints [-0.328, -70.049, -104.48, -5.471, 90.328, -90]
  MoveL 479 to (-601.31, -203, 860) mm, rotated rx 180 ry 0 rz -90 deg; joints [1.717, -71.17, -106.216, -2.614, 88.283, -90]
  MoveL 480 to (-604.11, -190.39, 864) mm, rotated rx 180 ry 0 rz -90 deg; joints [1.107, -70.705, -108.358, -0.937, 88.893, -90]
  MoveL 481 to (-605.51, -177.26, 866) mm, rotated rx 180 ry 0 rz -90 deg; joints [0.796, -70.5, -110.408, 0.907, 89.204, -90]
  MoveL 482 to (-606.91, -164.05, 868) mm, rotated rx 180 ry 0 rz -90 deg; joints [0.48, -70.356, -112.428, 2.784, 89.52, -90]
  MoveL 483 to (-612.5, -151.83, 876) mm, rotated rx 180 ry 0 rz -90 deg; joints [-0.826, -69.661, -114.654, 4.314, 90.826, -90]
  MoveL 484 to (-609, -137.3, 871) mm, rotated rx 180 ry 0 rz -90 deg; joints [-0.001, -70.375, -116.335, 6.711, 90.001, -90]
  MoveL 485 to (-611.1, -124.07, 874) mm, rotated rx 180 ry 0 rz -90 deg; joints [-0.493, -70.335, -118.311, 8.645, 90.493, -90]
  MoveL 486 to (-612.5, -110.62, 876) mm, rotated rx 180 ry 0 rz -90 deg; joints [-0.826, -70.478, -120.213, 10.691, 90.826, -90]
  MoveL 487 to (-609, -96.33, 871) mm, rotated rx 180 ry 0 rz -90 deg; joints [-0.001, -71.467, -121.714, 13.18, 90.001, -90]
  MoveL 488 to (-600.61, -81.53, 859) mm, rotated rx 180 ry 0 rz -90 deg; joints [1.867, -73.385, -122.677, 16.061, 88.133, -90]
  MoveL 489 to (-599.91, -67.98, 858) mm, rotated rx 180 ry 0 rz -90 deg; joints [2.016, -74.147, -124.227, 18.374, 87.984, -90]
  MoveL 490 to (-597.82, -54.34, 855) mm, rotated rx 180 ry 0 rz -90 deg; joints [2.456, -75.246, -125.576, 20.823, 87.544, -90]
  MoveL 491 to (-592.92, -40.59, 848) mm, rotated rx 180 ry 0 rz -90 deg; joints [3.449, -76.937, -126.527, 23.464, 86.551, -90]
  MoveL 492 to (-591.52, -27.23, 846) mm, rotated rx 180 ry 0 rz -90 deg; joints [3.724, -78.121, -127.795, 25.917, 86.276, -90]
  MoveL 493 to (-588.03, -13.88, 841) mm, rotated rx 180 ry 0 rz -90 deg; joints [4.395, -79.773, -128.721, 28.494, 85.605, -90]
  MoveL 494 to (-583.13, -0.69, 834) mm, rotated rx 180 ry 0 rz -90 deg; joints [5.297, -81.766, -129.347, 31.113, 84.703, -90]
  MoveL 495 to (-581.74, 12.36, 832) mm, rotated rx 180 ry 0 rz -90 deg; joints [5.547, -83.237, -130.378, 33.615, 84.453, -90]
  MoveL 496 to (-577.54, 25.22, 826) mm, rotated rx 180 ry 0 rz -90 deg; joints [6.276, -85.275, -130.899, 36.174, 83.724, -90]
  MoveL 497 to (-570.55, 37.71, 816) mm, rotated rx 180 ry 0 rz -90 deg; joints [7.428, -87.842, -130.839, 38.681, 82.572, -90]
  MoveL 498 to (-565.65, 50.08, 809) mm, rotated rx 180 ry 0 rz -90 deg; joints [8.189, -90.099, -130.992, 41.091, 81.811, -90]
  MoveL 499 to (-560.06, 62.14, 801) mm, rotated rx 180 ry 0 rz -90 deg; joints [9.017, -92.495, -130.896, 43.391, 80.983, -90]
  MoveL 500 to (-560.76, 74.8, 802) mm, rotated rx 180 ry 0 rz -90 deg; joints [8.916, -93.976, -131.884, 45.86, 81.084, -90]
  MoveL 501 to (-555.17, 86.5, 794) mm, rotated rx 180 ry 0 rz -90 deg; joints [9.706, -96.422, -131.59, 48.011, 80.294, -90]
  MoveL 502 to (-551.67, 98.33, 789) mm, rotated rx 180 ry 0 rz -90 deg; joints [10.179, -98.58, -131.603, 50.183, 79.821, -90]
  MoveL 503 to (-548.17, 110, 784) mm, rotated rx 180 ry 0 rz -90 deg; joints [10.637, -100.747, -131.528, 52.275, 79.363, -90]
  MoveL 504 to (-541.88, 120.89, 775) mm, rotated rx 180 ry 0 rz -90 deg; joints [11.426, -103.224, -130.773, 53.997, 78.574, -90]
  MoveL 505 to (-573.47, -487.49, 839) mm, rotated rx 180 ry 0 rz -90 deg; joints [7.444, -88.906, -45.632, -45.462, 82.556, -90]
  MoveL 506 to (-567.32, -469.24, 830) mm, rotated rx 180 ry 0 rz -90 deg; joints [8.468, -87.649, -50.515, -41.837, 81.532, -90]
  MoveL 507 to (-570.06, -458.43, 834) mm, rotated rx 180 ry 0 rz -90 deg; joints [8.021, -85.993, -54.128, -39.88, 81.979, -90]
  MoveL 508 to (-572.79, -447.49, 838) mm, rotated rx 180 ry 0 rz -90 deg; joints [7.561, -84.434, -57.559, -38.007, 82.439, -90]
  MoveL 509 to (-570.06, -432.27, 834) mm, rotated rx 180 ry 0 rz -90 deg; joints [8.021, -83.444, -61.179, -35.377, 81.979, -90]
  MoveL 510 to (-565.95, -416.18, 828) mm, rotated rx 180 ry 0 rz -90 deg; joints [8.687, -82.741, -64.606, -32.653, 81.313, -90]
  MoveL 511 to (-567.32, -404.17, 830) mm, rotated rx 180 ry 0 rz -90 deg; joints [8.468, -81.589, -67.62, -30.791, 81.532, -90]
  MoveL 512 to (-563.9, -388.79, 825) mm, rotated rx 180 ry 0 rz -90 deg; joints [9.01, -81.051, -70.637, -28.312, 80.99, -90]
  MoveL 513 to (-560.49, -373.58, 820) mm, rotated rx 180 ry 0 rz -90 deg; joints [9.532, -80.636, -73.468, -25.897, 80.468, -90]
  MoveL 514 to (-571.42, -367.76, 836) mm, rotated rx 180 ry 0 rz -90 deg; joints [7.793, -78.5, -76.081, -25.419, 82.207, -90]
  MoveL 515 to (-570.06, -353.8, 834) mm, rotated rx 180 ry 0 rz -90 deg; joints [8.021, -77.923, -78.756, -23.322, 81.979, -90]
  MoveL 516 to (-565.27, -337.86, 827) mm, rotated rx 180 ry 0 rz -90 deg; joints [8.795, -77.884, -81.296, -20.82, 81.205, -90]
  MoveL 517 to (-570.06, -327.64, 834) mm, rotated rx 180 ry 0 rz -90 deg; joints [8.021, -76.619, -83.829, -19.552, 81.979, -90]
  MoveL 518 to (-568.69, -313.81, 832) mm, rotated rx 180 ry 0 rz -90 deg; joints [8.246, -76.248, -86.23, -17.522, 81.754, -90]
  MoveL 519 to (-570.06, -301.49, 834) mm, rotated rx 180 ry 0 rz -90 deg; joints [8.021, -75.545, -88.618, -15.837, 81.979, -90]
  MoveL 520 to (-570.74, -288.76, 835) mm, rotated rx 180 ry 0 rz -90 deg; joints [7.907, -74.989, -90.94, -14.071, 82.093, -90]
  MoveL 521 to (-578.26, -279.29, 846) mm, rotated rx 180 ry 0 rz -90 deg; joints [6.599, -73.46, -93.427, -13.113, 83.401, -90]
  MoveL 522 to (-574.84, -264.45, 841) mm, rotated rx 180 ry 0 rz -90 deg; joints [7.207, -73.601, -95.545, -10.854, 82.793, -90]
  MoveL 523 to (-579.62, -253.36, 848) mm, rotated rx 180 ry 0 rz -90 deg; joints [6.35, -72.548, -97.907, -9.545, 83.65, -90]
  MoveL 524 to (-580.31, -240.34, 849) mm, rotated rx 180 ry 0 rz -90 deg; joints [6.224, -72.169, -100.082, -7.749, 83.776, -90]
  MoveL 525 to (-584.41, -228.63, 855) mm, rotated rx 180 ry 0 rz -90 deg; joints [5.448, -71.302, -102.375, -6.323, 84.552, -90]
  MoveL 526 to (-588.51, -216.74, 861) mm, rotated rx 180 ry 0 rz -90 deg; joints [4.637, -70.48, -104.65, -4.87, 85.363, -90]
  MoveL 527 to (-586.46, -202.53, 858) mm, rotated rx 180 ry 0 rz -90 deg; joints [5.047, -70.681, -106.601, -2.718, 84.953, -90]
  MoveL 528 to (-589.19, -189.95, 862) mm, rotated rx 180 ry 0 rz -90 deg; joints [4.499, -70.174, -108.761, -1.065, 85.501, -90]
  MoveL 529 to (-598.08, -179.1, 875) mm, rotated rx 180 ry 0 rz -90 deg; joints [2.599, -68.737, -111.237, -0.026, 87.401, -90]
  MoveL 530 to (-596.71, -165, 873) mm, rotated rx 180 ry 0 rz -90 deg; joints [2.903, -68.991, -113.141, 2.132, 87.097, -90]
  MoveL 531 to (-597.4, -151.48, 874) mm, rotated rx 180 ry 0 rz -90 deg; joints [2.752, -68.989, -115.118, 4.108, 87.248, -90]
  MoveL 532 to (-594.66, -137.15, 870) mm, rotated rx 180 ry 0 rz -90 deg; joints [3.352, -69.635, -116.823, 6.458, 86.649, -90]
  MoveL 533 to (-596.03, -123.79, 872) mm, rotated rx 180 ry 0 rz -90 deg; joints [3.054, -69.671, -118.768, 8.439, 86.946, -90]
  MoveL 534 to (-598.08, -110.49, 875) mm, rotated rx 180 ry 0 rz -90 deg; joints [2.599, -69.667, -120.738, 10.405, 87.401, -90]
  MoveL 535 to (-591.93, -95.78, 866) mm, rotated rx 180 ry 0 rz -90 deg; joints [3.934, -71.193, -121.973, 13.166, 86.066, -90]
  MoveL 536 to (-589.88, -81.91, 863) mm, rotated rx 180 ry 0 rz -90 deg; joints [4.359, -72.106, -123.471, 15.577, 85.641, -90]
  MoveL 537 to (-587.14, -68.06, 859) mm, rotated rx 180 ry 0 rz -90 deg; joints [4.912, -73.251, -124.824, 18.075, 85.088, -90]
  MoveL 538 to (-585.78, -54.46, 857) mm, rotated rx 180 ry 0 rz -90 deg; joints [5.182, -74.245, -126.253, 20.498, 84.818, -90]
  MoveL 539 to (-579.62, -40.59, 848) mm, rotated rx 180 ry 0 rz -90 deg; joints [6.35, -76.26, -127.019, 23.279, 83.65, -90]
  MoveL 540 to (-575.52, -27.1, 842) mm, rotated rx 180 ry 0 rz -90 deg; joints [7.087, -77.991, -127.914, 25.905, 82.913, -90]
  MoveL 541 to (-577.57, -13.95, 845) mm, rotated rx 180 ry 0 rz -90 deg; joints [6.723, -78.636, -129.585, 28.221, 83.277, -90]
  MoveL 542 to (-570.74, -0.69, 835) mm, rotated rx 180 ry 0 rz -90 deg; joints [7.907, -81.086, -129.899, 30.985, 82.093, -90]
  MoveL 543 to (-567.32, 12.33, 830) mm, rotated rx 180 ry 0 rz -90 deg; joints [8.468, -82.967, -130.601, 33.567, 81.532, -90]
  MoveL 544 to (-561.85, 25.1, 822) mm, rotated rx 180 ry 0 rz -90 deg; joints [9.325, -85.305, -130.851, 36.155, 80.675, -90]
  MoveL 545 to (-561.85, 37.99, 822) mm, rotated rx 180 ry 0 rz -90 deg; joints [9.325, -86.712, -131.946, 38.658, 80.675, -90]
  MoveL 546 to (-556.39, 50.39, 814) mm, rotated rx 180 ry 0 rz -90 deg; joints [10.135, -89.165, -131.977, 41.142, 79.865, -90]
  MoveL 547 to (-552.97, 62.76, 809) mm, rotated rx 180 ry 0 rz -90 deg; joints [10.618, -91.3, -132.275, 43.575, 79.382, -90]
  MoveL 548 to (-544.77, 74.33, 797) mm, rotated rx 180 ry 0 rz -90 deg; joints [11.713, -94.226, -131.509, 45.734, 78.287, -90]
  MoveL 549 to (-543.4, 86.61, 795) mm, rotated rx 180 ry 0 rz -90 deg; joints [11.887, -96.082, -132.013, 48.095, 78.113, -90]
  MoveL 550 to (-539.98, 98.45, 790) mm, rotated rx 180 ry 0 rz -90 deg; joints [12.311, -98.278, -132.009, 50.286, 77.689, -90]
  MoveL 551 to (-537.93, 110.42, 787) mm, rotated rx 180 ry 0 rz -90 deg; joints [12.559, -100.306, -132.212, 52.519, 77.441, -90]
  MoveL 552 to (-529.04, 120.74, 774) mm, rotated rx 180 ry 0 rz -90 deg; joints [13.579, -103.166, -130.817, 53.983, 76.421, -90]
  MoveL 553 to (-558.31, -485.75, 836) mm, rotated rx 180 ry 0 rz -90 deg; joints [10.558, -88.596, -46.294, -45.111, 79.442, -90]
  MoveL 554 to (-557.65, -472.07, 835) mm, rotated rx 180 ry 0 rz -90 deg; joints [10.66, -87.01, -50.554, -42.437, 79.34, -90]
  MoveL 555 to (-556.98, -458.43, 834) mm, rotated rx 180 ry 0 rz -90 deg; joints [10.76, -85.601, -54.479, -39.92, 79.24, -90]
  MoveL 556 to (-558.31, -446.42, 836) mm, rotated rx 180 ry 0 rz -90 deg; joints [10.558, -84.147, -58.004, -37.848, 79.442, -90]
  MoveL 557 to (-555.64, -431.23, 832) mm, rotated rx 180 ry 0 rz -90 deg; joints [10.959, -83.197, -61.573, -35.23, 79.041, -90]
  MoveL 558 to (-556.98, -419.19, 834) mm, rotated rx 180 ry 0 rz -90 deg; joints [10.76, -81.943, -64.742, -33.315, 79.24, -90]
  MoveL 559 to (-555.64, -405.14, 832) mm, rotated rx 180 ry 0 rz -90 deg; joints [10.959, -81.07, -67.875, -31.056, 79.041, -90]
  MoveL 560 to (-555.64, -392.09, 832) mm, rotated rx 180 ry 0 rz -90 deg; joints [10.959, -80.128, -70.824, -29.047, 79.041, -90]
  MoveL 561 to (-550.3, -375.4, 824) mm, rotated rx 180 ry 0 rz -90 deg; joints [11.726, -79.962, -73.708, -26.33, 78.274, -90]
  MoveL 562 to (-555.64, -366, 832) mm, rotated rx 180 ry 0 rz -90 deg; joints [10.959, -78.458, -76.397, -25.145, 79.041, -90]
  MoveL 563 to (-556.31, -353.38, 833) mm, rotated rx 180 ry 0 rz -90 deg; joints [10.86, -77.627, -79.045, -23.328, 79.14, -90]
  MoveL 564 to (-551.63, -337.45, 826) mm, rotated rx 180 ry 0 rz -90 deg; joints [11.539, -77.631, -81.551, -20.818, 78.461, -90]
  MoveL 565 to (-554.31, -326.07, 830) mm, rotated rx 180 ry 0 rz -90 deg; joints [11.155, -76.626, -84.067, -19.307, 78.845, -90]
  MoveL 566 to (-558.31, -315.32, 836) mm, rotated rx 180 ry 0 rz -90 deg; joints [10.558, -75.454, -86.572, -17.973, 79.442, -90]
  MoveL 567 to (-559.65, -302.93, 838) mm, rotated rx 180 ry 0 rz -90 deg; joints [10.353, -74.728, -88.98, -16.293, 79.647, -90]
  MoveL 568 to (-562.99, -291.52, 843) mm, rotated rx 180 ry 0 rz -90 deg; joints [9.827, -73.729, -91.403, -14.868, 80.173, -90]
  MoveL 569 to (-571, -282.26, 855) mm, rotated rx 180 ry 0 rz -90 deg; joints [8.478, -72.038, -93.933, -14.029, 81.522, -90]
  MoveL 570 to (-566.33, -266.66, 848) mm, rotated rx 180 ry 0 rz -90 deg; joints [9.28, -72.376, -96.047, -11.577, 80.72, -90]
  MoveL 571 to (-566.33, -253.36, 848) mm, rotated rx 180 ry 0 rz -90 deg; joints [9.28, -72.042, -98.244, -9.714, 80.72, -90]
  MoveL 572 to (-576.34, -244.31, 863) mm, rotated rx 180 ry 0 rz -90 deg; joints [7.506, -70.097, -100.836, -9.067, 82.494, -90]
  MoveL 573 to (-576.34, -230.77, 863) mm, rotated rx 180 ry 0 rz -90 deg; joints [7.506, -69.834, -102.997, -7.17, 82.494, -90]
  MoveL 574 to (-578.35, -218, 866) mm, rotated rx 180 ry 0 rz -90 deg; joints [7.125, -69.291, -105.21, -5.499, 82.875, -90]
  MoveL 575 to (-574.34, -203, 860) mm, rotated rx 180 ry 0 rz -90 deg; joints [7.877, -69.839, -107.065, -3.096, 82.123, -90]
  MoveL 576 to (-577.68, -190.62, 865) mm, rotated rx 180 ry 0 rz -90 deg; joints [7.253, -69.171, -109.289, -1.539, 82.747, -90]
  MoveL 577 to (-579.02, -177.46, 867) mm, rotated rx 180 ry 0 rz -90 deg; joints [6.996, -68.912, -111.369, 0.281, 83.004, -90]
  MoveL 578 to (-586.36, -165.94, 878) mm, rotated rx 180 ry 0 rz -90 deg; joints [5.508, -67.637, -113.815, 1.452, 84.492, -90]
  MoveL 579 to (-583.69, -151.48, 874) mm, rotated rx 180 ry 0 rz -90 deg; joints [6.064, -68.208, -115.59, 3.798, 83.936, -90]
  MoveL 580 to (-585.03, -138.09, 876) mm, rotated rx 180 ry 0 rz -90 deg; joints [5.788, -68.135, -117.595, 5.731, 84.212, -90]
  MoveL 581 to (-585.69, -124.5, 877) mm, rotated rx 180 ry 0 rz -90 deg; joints [5.649, -68.259, -119.52, 7.78, 84.352, -90]
  MoveL 582 to (-579.02, -109.48, 867) mm, rotated rx 180 ry 0 rz -90 deg; joints [6.996, -69.882, -120.755, 10.637, 83.004, -90]
  MoveL 583 to (-579.02, -95.89, 867) mm, rotated rx 180 ry 0 rz -90 deg; joints [6.996, -70.32, -122.509, 12.829, 83.004, -90]
  MoveL 584 to (-580.35, -82.48, 869) mm, rotated rx 180 ry 0 rz -90 deg; joints [6.735, -70.581, -124.362, 14.943, 83.265, -90]
  MoveL 585 to (-572.34, -67.9, 857) mm, rotated rx 180 ry 0 rz -90 deg; joints [8.24, -72.845, -125.12, 17.965, 81.76, -90]
  MoveL 586 to (-573.01, -54.53, 858) mm, rotated rx 180 ry 0 rz -90 deg; joints [8.12, -73.439, -126.79, 20.229, 81.88, -90]
  MoveL 587 to (-564.99, -40.5, 846) mm, rotated rx 180 ry 0 rz -90 deg; joints [9.501, -75.956, -127.252, 23.208, 80.499, -90]
  MoveL 588 to (-559.65, -26.97, 838) mm, rotated rx 180 ry 0 rz -90 deg; joints [10.353, -78.024, -127.91, 25.934, 79.647, -90]
  MoveL 589 to (-562.99, -13.92, 843) mm, rotated rx 180 ry 0 rz -90 deg; joints [9.827, -78.357, -129.801, 28.158, 80.173, -90]
  MoveL 590 to (-562.99, -0.7, 843) mm, rotated rx 180 ry 0 rz -90 deg; joints [9.827, -79.507, -131.141, 30.648, 80.173, -90]
  MoveL 591 to (-554.97, 12.35, 831) mm, rotated rx 180 ry 0 rz -90 deg; joints [11.058, -82.401, -131.076, 33.476, 78.942, -90]
  MoveL 592 to (-553.64, 25.32, 829) mm, rotated rx 180 ry 0 rz -90 deg; joints [11.252, -84.007, -132.025, 36.032, 78.748, -90]
  MoveL 593 to (-544.96, 37.71, 816) mm, rotated rx 180 ry 0 rz -90 deg; joints [12.448, -87.124, -131.513, 38.637, 77.552, -90]
  MoveL 594 to (-540.95, 50.14, 810) mm, rotated rx 180 ry 0 rz -90 deg; joints [12.963, -89.357, -131.74, 41.098, 77.037, -90]
  MoveL 595 to (-540.28, 62.76, 809) mm, rotated rx 180 ry 0 rz -90 deg; joints [13.047, -91.033, -132.55, 43.583, 76.953, -90]
  MoveL 596 to (-536.27, 74.89, 803) mm, rotated rx 180 ry 0 rz -90 deg; joints [13.537, -93.354, -132.587, 45.941, 76.463, -90]
  MoveL 597 to (-530.93, 86.61, 795) mm, rotated rx 180 ry 0 rz -90 deg; joints [14.158, -95.899, -132.227, 48.126, 75.842, -90]
  MoveL 598 to (-529.6, 98.83, 793) mm, rotated rx 180 ry 0 rz -90 deg; joints [14.309, -97.827, -132.652, 50.479, 75.692, -90]
  MoveL 599 to (-526.92, 110.7, 789) mm, rotated rx 180 ry 0 rz -90 deg; joints [14.602, -99.987, -132.7, 52.686, 75.398, -90]
  MoveL 600 to (-526.26, 122.92, 788) mm, rotated rx 180 ry 0 rz -90 deg; joints [14.675, -101.911, -133.129, 55.04, 75.325, -90]
  MoveL 601 to (-545.2, -485.75, 836) mm, rotated rx 180 ry 0 rz -90 deg; joints [13.329, -88.26, -46.615, -45.125, 76.671, -90]
  MoveL 602 to (-544.55, -472.07, 835) mm, rotated rx 180 ry 0 rz -90 deg; joints [13.416, -86.687, -50.851, -42.463, 76.584, -90]
  MoveL 603 to (-546.51, -460.63, 838) mm, rotated rx 180 ry 0 rz -90 deg; joints [13.152, -85.039, -54.556, -40.405, 76.848, -90]
  MoveL 604 to (-547.16, -448.02, 839) mm, rotated rx 180 ry 0 rz -90 deg; joints [13.063, -83.626, -58.152, -38.222, 76.937, -90]
  MoveL 605 to (-539.99, -429.16, 828) mm, rotated rx 180 ry 0 rz -90 deg; joints [14.009, -83.201, -61.939, -34.86, 75.991, -90]
  MoveL 606 to (-541.94, -417.68, 831) mm, rotated rx 180 ry 0 rz -90 deg; joints [13.759, -81.872, -65.063, -33.065, 76.241, -90]
  MoveL 607 to (-541.29, -404.17, 830) mm, rotated rx 180 ry 0 rz -90 deg; joints [13.843, -80.941, -68.144, -30.915, 76.157, -90]
  MoveL 608 to (-544.55, -393.51, 835) mm, rotated rx 180 ry 0 rz -90 deg; joints [13.416, -79.571, -71.023, -29.406, 76.584, -90]
  MoveL 609 to (-545.2, -380.87, 836) mm, rotated rx 180 ry 0 rz -90 deg; joints [13.329, -78.6, -73.867, -27.533, 76.671, -90]
  MoveL 610 to (-541.94, -365.56, 831) mm, rotated rx 180 ry 0 rz -90 deg; joints [13.759, -78.254, -76.623, -25.123, 76.241, -90]
  MoveL 611 to (-542.59, -352.95, 832) mm, rotated rx 180 ry 0 rz -90 deg; joints [13.674, -77.42, -79.267, -23.313, 76.326, -90]
  MoveL 612 to (-541.29, -339.09, 830) mm, rotated rx 180 ry 0 rz -90 deg; joints [13.843, -76.946, -81.805, -21.249, 76.157, -90]
  MoveL 613 to (-543.9, -327.64, 834) mm, rotated rx 180 ry 0 rz -90 deg; joints [13.503, -75.911, -84.343, -19.746, 76.497, -90]
  MoveL 614 to (-543.9, -314.57, 834) mm, rotated rx 180 ry 0 rz -90 deg; joints [13.503, -75.341, -86.769, -17.89, 76.497, -90]
  MoveL 615 to (-547.81, -303.66, 840) mm, rotated rx 180 ry 0 rz -90 deg; joints [12.973, -74.167, -89.261, -16.573, 77.027, -90]
  MoveL 616 to (-551.73, -292.56, 846) mm, rotated rx 180 ry 0 rz -90 deg; joints [12.416, -73.023, -91.725, -15.251, 77.584, -90]
  MoveL 617 to (-554.33, -280.61, 850) mm, rotated rx 180 ry 0 rz -90 deg; joints [12.03, -72.133, -94.119, -13.748, 77.97, -90]
  MoveL 618 to (-556.29, -268.23, 853) mm, rotated rx 180 ry 0 rz -90 deg; joints [11.732, -71.391, -96.459, -12.15, 78.268, -90]
  MoveL 619 to (-553.68, -253.66, 849) mm, rotated rx 180 ry 0 rz -90 deg; joints [12.128, -71.505, -98.552, -9.943, 77.872, -90]
  MoveL 620 to (-555.64, -241.19, 852) mm, rotated rx 180 ry 0 rz -90 deg; joints [11.833, -70.859, -100.813, -8.328, 78.168, -90]
  MoveL 621 to (-564.77, -231.58, 866) mm, rotated rx 180 ry 0 rz -90 deg; joints [10.352, -68.944, -103.426, -7.63, 79.648, -90]
  MoveL 622 to (-568.68, -219.51, 872) mm, rotated rx 180 ry 0 rz -90 deg; joints [9.663, -68.011, -105.761, -6.228, 80.337, -90]
  MoveL 623 to (-561.51, -203.24, 861) mm, rotated rx 180 ry 0 rz -90 deg; joints [10.901, -69.186, -107.436, -3.378, 79.099, -90]
  MoveL 624 to (-566.72, -191.5, 869) mm, rotated rx 180 ry 0 rz -90 deg; joints [10.012, -68.094, -109.813, -2.093, 79.988, -90]
  MoveL 625 to (-565.42, -177.46, 867) mm, rotated rx 180 ry 0 rz -90 deg; joints [10.24, -68.312, -111.732, 0.044, 79.76, -90]
  MoveL 626 to (-573.25, -166.13, 879) mm, rotated rx 180 ry 0 rz -90 deg; joints [8.813, -66.803, -114.271, 1.074, 81.187, -90]
  MoveL 627 to (-570.64, -151.66, 875) mm, rotated rx 180 ry 0 rz -90 deg; joints [9.305, -67.398, -116.043, 3.441, 80.695, -90]
  MoveL 628 to (-572.59, -138.41, 878) mm, rotated rx 180 ry 0 rz -90 deg; joints [8.938, -67.162, -118.12, 5.282, 81.062, -90]
  MoveL 629 to (-568.68, -123.79, 872) mm, rotated rx 180 ry 0 rz -90 deg; joints [9.663, -68.211, -119.654, 7.865, 80.337, -90]
  MoveL 630 to (-568.03, -109.99, 871) mm, rotated rx 180 ry 0 rz -90 deg; joints [9.781, -68.683, -121.412, 10.095, 80.219, -90]
  MoveL 631 to (-564.77, -95.78, 866) mm, rotated rx 180 ry 0 rz -90 deg; joints [10.352, -69.816, -122.839, 12.655, 79.648, -90]
  MoveL 632 to (-567.38, -82.57, 870) mm, rotated rx 180 ry 0 rz -90 deg; joints [9.897, -69.765, -124.854, 14.619, 80.103, -90]
  MoveL 633 to (-562.16, -68.3, 862) mm, rotated rx 180 ry 0 rz -90 deg; joints [10.793, -71.546, -125.907, 17.452, 79.207, -90]
  MoveL 634 to (-561.51, -54.72, 861) mm, rotated rx 180 ry 0 rz -90 deg; joints [10.901, -72.419, -127.435, 19.854, 79.099, -90]
  MoveL 635 to (-554.99, -40.74, 851) mm, rotated rx 180 ry 0 rz -90 deg; joints [11.932, -74.737, -128.071, 22.808, 78.068, -90]
  MoveL 636 to (-548.46, -27.07, 841) mm, rotated rx 180 ry 0 rz -90 deg; joints [12.882, -77.167, -128.53, 25.697, 77.118, -90]
  MoveL 637 to (-545.2, -13.8, 836) mm, rotated rx 180 ry 0 rz -90 deg; joints [13.329, -78.947, -129.373, 28.32, 76.671, -90]
  MoveL 638 to (-547.81, -0.69, 840) mm, rotated rx 180 ry 0 rz -90 deg; joints [12.973, -79.501, -131.146, 30.647, 77.027, -90]
  MoveL 639 to (-541.29, 12.33, 830) mm, rotated rx 180 ry 0 rz -90 deg; joints [13.843, -82.194, -131.244, 33.438, 76.157, -90]
  MoveL 640 to (-543.9, 25.47, 834) mm, rotated rx 180 ry 0 rz -90 deg; joints [13.503, -82.976, -132.927, 35.903, 76.497, -90]
  MoveL 641 to (-537.38, 38.08, 824) mm, rotated rx 180 ry 0 rz -90 deg; joints [14.334, -85.8, -132.793, 38.593, 75.666, -90]
  MoveL 642 to (-532.16, 50.51, 816) mm, rotated rx 180 ry 0 rz -90 deg; joints [14.954, -88.374, -132.768, 41.142, 75.046, -90]
  MoveL 643 to (-530.2, 63.07, 813) mm, rotated rx 180 ry 0 rz -90 deg; joints [15.177, -90.343, -133.315, 43.658, 74.823, -90]
  MoveL 644 to (-523.03, 74.8, 802) mm, rotated rx 180 ry 0 rz -90 deg; joints [15.954, -93.309, -132.617, 45.926, 74.046, -90]
  MoveL 645 to (-518.46, 86.61, 795) mm, rotated rx 180 ry 0 rz -90 deg; joints [16.417, -95.776, -132.37, 48.146, 73.583, -90]
  MoveL 646 to (-519.77, 99.33, 797) mm, rotated rx 180 ry 0 rz -90 deg; joints [16.287, -97.309, -133.401, 50.71, 73.713, -90]
  MoveL 647 to (-516.51, 111.12, 792) mm, rotated rx 180 ry 0 rz -90 deg; joints [16.608, -99.613, -133.289, 52.902, 73.392, -90]
  MoveL 648 to (-515.2, 123.23, 790) mm, rotated rx 180 ry 0 rz -90 deg; joints [16.734, -101.657, -133.562, 55.218, 73.266, -90]
  MoveL 649 to (-537.19, -490.39, 844) mm, rotated rx 180 ry 0 rz -90 deg; joints [15.487, -87.596, -46.272, -46.132, 74.513, -90]
  MoveL 650 to (-534, -474.33, 839) mm, rotated rx 180 ry 0 rz -90 deg; joints [15.869, -86.203, -50.841, -42.956, 74.131, -90]
  MoveL 651 to (-530.82, -458.43, 834) mm, rotated rx 180 ry 0 rz -90 deg; joints [16.237, -85.055, -54.962, -39.983, 73.763, -90]
  MoveL 652 to (-534, -448.02, 839) mm, rotated rx 180 ry 0 rz -90 deg; joints [15.869, -83.371, -58.368, -38.261, 74.131, -90]
  MoveL 653 to (-527, -429.16, 828) mm, rotated rx 180 ry 0 rz -90 deg; joints [16.658, -83, -62.108, -34.892, 73.342, -90]
  MoveL 654 to (-529.55, -418.19, 832) mm, rotated rx 180 ry 0 rz -90 deg; joints [16.379, -81.573, -65.218, -33.208, 73.621, -90]
  MoveL 655 to (-529.55, -405.14, 832) mm, rotated rx 180 ry 0 rz -90 deg; joints [16.379, -80.554, -68.286, -31.16, 73.621, -90]
  MoveL 656 to (-528.91, -391.62, 831) mm, rotated rx 180 ry 0 rz -90 deg; joints [16.45, -79.704, -71.235, -29.061, 73.55, -90]
  MoveL 657 to (-528.27, -378.14, 830) mm, rotated rx 180 ry 0 rz -90 deg; joints [16.52, -78.934, -74.061, -27.005, 73.48, -90]
  MoveL 658 to (-534.64, -369.52, 840) mm, rotated rx 180 ry 0 rz -90 deg; joints [15.794, -77.153, -76.802, -26.045, 74.206, -90]
  MoveL 659 to (-530.82, -353.8, 834) mm, rotated rx 180 ry 0 rz -90 deg; joints [16.237, -76.992, -79.448, -23.56, 73.763, -90]
  MoveL 660 to (-530.18, -340.31, 833) mm, rotated rx 180 ry 0 rz -90 deg; joints [16.308, -76.411, -82.005, -21.584, 73.692, -90]
  MoveL 661 to (-532.09, -328.43, 836) mm, rotated rx 180 ry 0 rz -90 deg; joints [16.092, -75.458, -84.546, -19.997, 73.908, -90]
  MoveL 662 to (-534, -316.45, 839) mm, rotated rx 180 ry 0 rz -90 deg; joints [15.869, -74.544, -87.04, -18.416, 74.131, -90]
  MoveL 663 to (-531.46, -301.85, 835) mm, rotated rx 180 ry 0 rz -90 deg; joints [16.164, -74.471, -89.324, -16.205, 73.836, -90]
  MoveL 664 to (-534, -290.14, 839) mm, rotated rx 180 ry 0 rz -90 deg; joints [15.869, -73.532, -91.747, -14.721, 74.131, -90]
  MoveL 665 to (-538.46, -279.29, 846) mm, rotated rx 180 ry 0 rz -90 deg; joints [15.33, -72.27, -94.227, -13.503, 74.67, -90]
  MoveL 666 to (-544.19, -268.86, 855) mm, rotated rx 180 ry 0 rz -90 deg; joints [14.587, -70.796, -96.746, -12.458, 75.413, -90]
  MoveL 667 to (-540.37, -253.66, 849) mm, rotated rx 180 ry 0 rz -90 deg; joints [15.088, -71.169, -98.77, -10.061, 74.912, -90]
  MoveL 668 to (-545.46, -242.61, 857) mm, rotated rx 180 ry 0 rz -90 deg; joints [14.414, -69.874, -101.227, -8.9, 75.586, -90]
  MoveL 669 to (-548.01, -230.24, 861) mm, rotated rx 180 ry 0 rz -90 deg; joints [14.059, -69.109, -103.522, -7.368, 75.941, -90]
  MoveL 670 to (-553.1, -218.75, 869) mm, rotated rx 180 ry 0 rz -90 deg; joints [13.311, -67.875, -105.952, -6.173, 76.689, -90]
  MoveL 671 to (-553.1, -205.12, 869) mm, rotated rx 180 ry 0 rz -90 deg; joints [13.311, -67.7, -108.053, -4.247, 76.689, -90]
  MoveL 672 to (-553.1, -191.5, 869) mm, rotated rx 180 ry 0 rz -90 deg; joints [13.311, -67.589, -110.111, -2.3, 76.689, -90]
  MoveL 673 to (-554.37, -178.28, 871) mm, rotated rx 180 ry 0 rz -90 deg; joints [13.115, -67.273, -112.226, -0.501, 76.885, -90]
  MoveL 674 to (-558.19, -165.75, 877) mm, rotated rx 180 ry 0 rz -90 deg; joints [12.507, -66.467, -114.518, 0.985, 77.493, -90]
  MoveL 675 to (-554.37, -150.96, 871) mm, rotated rx 180 ry 0 rz -90 deg; joints [13.115, -67.38, -116.155, 3.535, 76.885, -90]
  MoveL 676 to (-553.73, -137.15, 870) mm, rotated rx 180 ry 0 rz -90 deg; joints [13.214, -67.689, -117.998, 5.687, 76.786, -90]
  MoveL 677 to (-555.64, -123.93, 873) mm, rotated rx 180 ry 0 rz -90 deg; joints [12.916, -67.496, -120.053, 7.55, 77.084, -90]
  MoveL 678 to (-556.92, -110.49, 875) mm, rotated rx 180 ry 0 rz -90 deg; joints [12.713, -67.523, -122.021, 9.545, 77.287, -90]
  MoveL 679 to (-556.92, -96.77, 875) mm, rotated rx 180 ry 0 rz -90 deg; joints [12.713, -67.931, -123.823, 11.753, 77.287, -90]
  MoveL 680 to (-554.37, -82.67, 871) mm, rotated rx 180 ry 0 rz -90 deg; joints [13.115, -69.042, -125.278, 14.32, 76.885, -90]
  MoveL 681 to (-545.46, -67.9, 857) mm, rotated rx 180 ry 0 rz -90 deg; joints [14.414, -71.825, -125.788, 17.613, 75.586, -90]
  MoveL 682 to (-545.46, -54.46, 857) mm, rotated rx 180 ry 0 rz -90 deg; joints [14.414, -72.551, -127.388, 19.94, 75.586, -90]
  MoveL 683 to (-544.19, -40.93, 855) mm, rotated rx 180 ry 0 rz -90 deg; joints [14.587, -73.697, -128.749, 22.445, 75.413, -90]
  MoveL 684 to (-535.28, -27.07, 841) mm, rotated rx 180 ry 0 rz -90 deg; joints [15.718, -76.835, -128.773, 25.607, 74.282, -90]
  MoveL 685 to (-534, -13.85, 839) mm, rotated rx 180 ry 0 rz -90 deg; joints [15.869, -78.185, -129.941, 28.126, 74.131, -90]
  MoveL 686 to (-530.18, -0.69, 833) mm, rotated rx 180 ry 0 rz -90 deg; joints [16.308, -80.25, -130.564, 30.814, 73.692, -90]
  MoveL 687 to (-530.18, 12.37, 833) mm, rotated rx 180 ry 0 rz -90 deg; joints [16.308, -81.492, -131.824, 33.316, 73.692, -90]
  MoveL 688 to (-530.82, 25.47, 834) mm, rotated rx 180 ry 0 rz -90 deg; joints [16.237, -82.7, -133.157, 35.857, 73.763, -90]
  MoveL 689 to (-516.18, 37.48, 811) mm, rotated rx 180 ry 0 rz -90 deg; joints [17.749, -87.413, -131.2, 38.613, 72.251, -90]
  MoveL 690 to (-516.18, 50.2, 811) mm, rotated rx 180 ry 0 rz -90 deg; joints [17.749, -88.885, -132.214, 41.099, 72.251, -90]
  MoveL 691 to (-513.64, 62.61, 807) mm, rotated rx 180 ry 0 rz -90 deg; joints [17.986, -90.969, -132.585, 43.553, 72.014, -90]
  MoveL 692 to (-507.27, 74.33, 797) mm, rotated rx 180 ry 0 rz -90 deg; joints [18.547, -93.821, -131.958, 45.779, 71.453, -90]
  MoveL 693 to (-504.09, 86.28, 792) mm, rotated rx 180 ry 0 rz -90 deg; joints [18.813, -96.054, -131.974, 48.028, 71.187, -90]
  MoveL 694 to (-506, 99.08, 795) mm, rotated rx 180 ry 0 rz -90 deg; joints [18.655, -97.454, -133.167, 50.621, 71.345, -90]
  MoveL 695 to (-504.73, 111.26, 793) mm, rotated rx 180 ry 0 rz -90 deg; joints [18.761, -99.47, -133.509, 52.979, 71.239, -90]
  MoveL 696 to (-500.91, 122.76, 787) mm, rotated rx 180 ry 0 rz -90 deg; joints [19.069, -101.883, -133.128, 55.011, 70.931, -90]
  MoveL 697 to (-520.85, -487.49, 839) mm, rotated rx 180 ry 0 rz -90 deg; joints [18.656, -87.668, -46.813, -45.519, 71.344, -90]
  MoveL 698 to (-518.98, -472.64, 836) mm, rotated rx 180 ry 0 rz -90 deg; joints [18.833, -86.221, -51.162, -42.617, 71.167, -90]
  MoveL 699 to (-517.74, -458.43, 834) mm, rotated rx 180 ry 0 rz -90 deg; joints [18.948, -84.903, -55.095, -40.002, 71.052, -90]
  MoveL 700 to (-517.12, -444.82, 833) mm, rotated rx 180 ry 0 rz -90 deg; joints [19.005, -83.66, -58.717, -37.623, 70.995, -90]
  MoveL 701 to (-520.23, -434.34, 838) mm, rotated rx 180 ry 0 rz -90 deg; joints [18.715, -82.043, -61.971, -35.986, 71.285, -90]
  MoveL 702 to (-518.36, -419.7, 835) mm, rotated rx 180 ry 0 rz -90 deg; joints [18.891, -81.17, -65.28, -33.55, 71.109, -90]
  MoveL 703 to (-524.57, -411.47, 845) mm, rotated rx 180 ry 0 rz -90 deg; joints [18.289, -79.243, -68.216, -32.541, 71.711, -90]
  MoveL 704 to (-517.74, -393.04, 834) mm, rotated rx 180 ry 0 rz -90 deg; joints [18.948, -79.279, -71.328, -29.394, 71.052, -90]
  MoveL 705 to (-516.5, -379.05, 832) mm, rotated rx 180 ry 0 rz -90 deg; joints [19.062, -78.601, -74.166, -27.233, 70.938, -90]
  MoveL 706 to (-518.98, -367.76, 836) mm, rotated rx 180 ry 0 rz -90 deg; joints [18.833, -77.383, -76.919, -25.699, 71.167, -90]
  MoveL 707 to (-518.98, -354.65, 836) mm, rotated rx 180 ry 0 rz -90 deg; joints [18.833, -76.627, -79.579, -23.794, 71.167, -90]
  MoveL 708 to (-517.12, -340.31, 833) mm, rotated rx 180 ry 0 rz -90 deg; joints [19.005, -76.263, -82.112, -21.625, 70.995, -90]
  MoveL 709 to (-517.74, -327.64, 834) mm, rotated rx 180 ry 0 rz -90 deg; joints [18.948, -75.522, -84.622, -19.856, 71.052, -90]
  MoveL 710 to (-520.85, -316.45, 839) mm, rotated rx 180 ry 0 rz -90 deg; joints [18.656, -74.365, -87.164, -18.471, 71.344, -90]
  MoveL 711 to (-522.09, -304.02, 841) mm, rotated rx 180 ry 0 rz -90 deg; joints [18.536, -73.592, -89.6, -16.808, 71.464, -90]
  MoveL 712 to (-520.23, -289.79, 838) mm, rotated rx 180 ry 0 rz -90 deg; joints [18.715, -73.473, -91.839, -14.688, 71.285, -90]
  MoveL 713 to (-523.33, -278.3, 843) mm, rotated rx 180 ry 0 rz -90 deg; joints [18.413, -72.422, -94.275, -13.303, 71.587, -90]
  MoveL 714 to (-527.68, -267.28, 850) mm, rotated rx 180 ry 0 rz -90 deg; joints [17.968, -71.148, -96.756, -12.096, 72.032, -90]
  MoveL 715 to (-525.81, -253.06, 847) mm, rotated rx 180 ry 0 rz -90 deg; joints [18.162, -71.187, -98.847, -9.966, 71.838, -90]
  MoveL 716 to (-532.02, -242.61, 857) mm, rotated rx 180 ry 0 rz -90 deg; joints [17.494, -69.58, -101.409, -9.011, 72.506, -90]
  MoveL 717 to (-532.64, -229.44, 858) mm, rotated rx 180 ry 0 rz -90 deg; joints [17.424, -69.185, -103.594, -7.221, 72.576, -90]
  MoveL 718 to (-529.54, -214.72, 853) mm, rotated rx 180 ry 0 rz -90 deg; joints [17.769, -69.669, -105.456, -4.875, 72.232, -90]
  MoveL 719 to (-541.95, -206.07, 873) mm, rotated rx 180 ry 0 rz -90 deg; joints [16.292, -66.764, -108.458, -4.779, 73.708, -90]
  MoveL 720 to (-538.85, -191.28, 868) mm, rotated rx 180 ry 0 rz -90 deg; joints [16.687, -67.334, -110.292, -2.373, 73.313, -90]
  MoveL 721 to (-538.23, -177.46, 867) mm, rotated rx 180 ry 0 rz -90 deg; joints [16.764, -67.43, -112.254, -0.316, 73.236, -90]
  MoveL 722 to (-545.06, -165.94, 878) mm, rotated rx 180 ry 0 rz -90 deg; joints [15.878, -65.849, -114.838, 0.687, 74.122, -90]
  MoveL 723 to (-540.71, -150.96, 871) mm, rotated rx 180 ry 0 rz -90 deg; joints [16.452, -66.95, -116.404, 3.354, 73.548, -90]
  MoveL 724 to (-543.2, -137.93, 875) mm, rotated rx 180 ry 0 rz -90 deg; joints [16.129, -66.501, -118.567, 5.068, 73.872, -90]
  MoveL 725 to (-548.78, -125.49, 884) mm, rotated rx 180 ry 0 rz -90 deg; joints [15.354, -65.349, -121.034, 6.382, 74.646, -90]
  MoveL 726 to (-543.2, -110.49, 875) mm, rotated rx 180 ry 0 rz -90 deg; joints [16.129, -67.039, -122.3, 9.34, 73.872, -90]
  MoveL 727 to (-544.44, -96.99, 877) mm, rotated rx 180 ry 0 rz -90 deg; joints [15.962, -67.122, -124.257, 11.379, 74.038, -90]
  MoveL 728 to (-538.23, -82.29, 867) mm, rotated rx 180 ry 0 rz -90 deg; joints [16.764, -69.231, -125.221, 14.452, 73.236, -90]
  MoveL 729 to (-543.2, -69.33, 875) mm, rotated rx 180 ry 0 rz -90 deg; joints [16.128, -68.532, -127.6, 16.132, 73.872, -90]
  MoveL 730 to (-533.88, -54.65, 860) mm, rotated rx 180 ry 0 rz -90 deg; joints [17.282, -71.71, -127.903, 19.613, 72.718, -90]
  MoveL 731 to (-526.43, -40.59, 848) mm, rotated rx 180 ry 0 rz -90 deg; joints [18.098, -74.52, -128.243, 22.763, 71.902, -90]
  MoveL 732 to (-520.85, -27.01, 839) mm, rotated rx 180 ry 0 rz -90 deg; joints [18.656, -76.931, -128.713, 25.644, 71.344, -90]
  MoveL 733 to (-517.12, -13.75, 833) mm, rotated rx 180 ry 0 rz -90 deg; joints [19.005, -78.937, -129.389, 28.326, 70.995, -90]
  MoveL 734 to (-518.36, -0.69, 835) mm, rotated rx 180 ry 0 rz -90 deg; joints [18.891, -79.753, -130.952, 30.705, 71.109, -90]
  MoveL 735 to (-520.85, 12.46, 839) mm, rotated rx 180 ry 0 rz -90 deg; joints [18.656, -80.375, -132.729, 33.104, 71.344, -90]
  MoveL 736 to (-517.74, 25.47, 834) mm, rotated rx 180 ry 0 rz -90 deg; joints [18.948, -82.519, -133.307, 35.826, 71.052, -90]
  MoveL 737 to (-507.81, 37.81, 818) mm, rotated rx 180 ry 0 rz -90 deg; joints [19.806, -86.342, -132.251, 38.593, 70.194, -90]
  MoveL 738 to (-505.33, 50.39, 814) mm, rotated rx 180 ry 0 rz -90 deg; joints [20.004, -88.409, -132.71, 41.119, 69.996, -90]
  MoveL 739 to (-499.74, 62.45, 805) mm, rotated rx 180 ry 0 rz -90 deg; joints [20.427, -91.19, -132.326, 43.516, 69.573, -90]
  MoveL 740 to (-496.64, 74.61, 800) mm, rotated rx 180 ry 0 rz -90 deg; joints [20.65, -93.444, -132.43, 45.874, 69.35, -90]
  MoveL 741 to (-491.05, 86.17, 791) mm, rotated rx 180 ry 0 rz -90 deg; joints [21.031, -96.18, -131.803, 47.983, 68.969, -90]
  MoveL 742 to (-490.43, 98.45, 790) mm, rotated rx 180 ry 0 rz -90 deg; joints [21.072, -97.996, -132.358, 50.354, 68.928, -90]
  MoveL 743 to (-489.81, 110.7, 789) mm, rotated rx 180 ry 0 rz -90 deg; joints [21.113, -99.876, -132.845, 52.721, 68.887, -90]
  MoveL 744 to (-488.57, 122.76, 787) mm, rotated rx 180 ry 0 rz -90 deg; joints [21.193, -101.905, -133.098, 55.003, 68.807, -90]
  MoveL 745 to (-508.9, -488.65, 841) mm, rotated rx 180 ry 0 rz -90 deg; joints [21.319, -87.452, -46.772, -45.776, 68.681, -90]
  MoveL 746 to (-507.69, -474.33, 839) mm, rotated rx 180 ry 0 rz -90 deg; joints [21.409, -85.933, -51.083, -42.984, 68.591, -90]
  MoveL 747 to (-504.06, -457.88, 833) mm, rotated rx 180 ry 0 rz -90 deg; joints [21.667, -84.909, -55.194, -39.896, 68.333, -90]
  MoveL 748 to (-508.3, -448.55, 840) mm, rotated rx 180 ry 0 rz -90 deg; joints [21.364, -83.027, -58.556, -38.417, 68.636, -90]
  MoveL 749 to (-510.11, -436.94, 843) mm, rotated rx 180 ry 0 rz -90 deg; joints [21.229, -81.535, -61.912, -36.553, 68.771, -90]
  MoveL 750 to (-499.82, -415.17, 826) mm, rotated rx 180 ry 0 rz -90 deg; joints [21.953, -81.932, -65.451, -32.617, 68.047, -90]
  MoveL 751 to (-508.3, -409.04, 840) mm, rotated rx 180 ry 0 rz -90 deg; joints [21.364, -79.591, -68.37, -32.039, 68.636, -90]
  MoveL 752 to (-504.66, -393.04, 834) mm, rotated rx 180 ry 0 rz -90 deg; joints [21.625, -79.21, -71.381, -29.41, 68.375, -90]
  MoveL 753 to (-503.45, -379.05, 832) mm, rotated rx 180 ry 0 rz -90 deg; joints [21.709, -78.539, -74.213, -27.248, 68.291, -90]
  MoveL 754 to (-505.87, -367.76, 836) mm, rotated rx 180 ry 0 rz -90 deg; joints [21.54, -77.304, -76.976, -25.72, 68.46, -90]
  MoveL 755 to (-504.66, -353.8, 834) mm, rotated rx 180 ry 0 rz -90 deg; joints [21.625, -76.77, -79.61, -23.62, 68.375, -90]
  MoveL 756 to (-504.66, -340.72, 834) mm, rotated rx 180 ry 0 rz -90 deg; joints [21.625, -76.082, -82.179, -21.74, 68.375, -90]
  MoveL 757 to (-503.45, -326.86, 832) mm, rotated rx 180 ry 0 rz -90 deg; joints [21.709, -75.689, -84.625, -19.686, 68.291, -90]
  MoveL 758 to (-510.11, -317.96, 843) mm, rotated rx 180 ry 0 rz -90 deg; joints [21.229, -73.792, -87.325, -18.883, 68.771, -90]
  MoveL 759 to (-511.93, -305.83, 846) mm, rotated rx 180 ry 0 rz -90 deg; joints [21.089, -72.874, -89.807, -17.319, 68.911, -90]
